C05453=1021.011,30.378,396.099,166.914,51.135,159.364
C05454=1021.017,30.627,396.085,166.917,51.129,159.363
C05455=1021.022,30.877,396.069,166.919,51.125,159.363
C05456=1021.028,31.126,396.055,166.923,51.119,159.362
C05457=1021.034,31.376,396.039,166.924,51.114,159.361
C05458=1021.040,31.626,396.024,166.928,51.109,159.361
C05459=1021.045,31.875,396.009,166.931,51.103,159.361
C05460=1021.051,32.124,395.993,166.933,51.098,159.360
C05461=1021.057,32.373,395.978,166.936,51.093,159.359
C05462=1021.062,32.623,395.962,166.938,51.088,159.359
C05463=1021.069,32.873,395.948,166.941,51.082,159.358
C05464=1021.074,33.122,395.932,166.944,51.077,159.358
C05465=1021.080,33.372,395.917,166.946,51.072,159.357
C05466=1021.086,33.621,395.901,166.949,51.066,159.357
C05467=1021.092,33.870,395.887,166.951,51.061,159.356
C05468=1021.098,34.120,395.871,166.954,51.056,159.356
C05469=1021.103,34.370,395.855,166.957,51.050,159.355
C05470=1021.109,34.619,395.841,166.959,51.045,159.355
C05471=1021.115,34.868,395.825,166.962,51.040,159.354
C05472=1021.121,35.117,395.810,166.964,51.035,159.353
C05473=1021.126,35.367,395.795,166.967,51.030,159.353
C05474=1021.133,35.617,395.780,166.970,51.024,159.352
C05475=1021.138,35.866,395.764,166.972,51.019,159.352
C05476=1021.144,36.116,395.748,166.975,51.013,159.351
C05477=1021.150,36.365,395.733,166.977,51.008,159.351
C05478=1021.156,36.615,395.718,166.980,51.002,159.350
C05479=1021.162,36.864,395.703,166.983,50.997,159.350
C05480=1021.168,37.113,395.687,166.985,50.992,159.349
C05481=1021.173,37.363,395.671,166.988,50.986,159.348
C05482=1021.178,37.613,395.656,166.990,50.982,159.348
C05483=1021.184,37.862,395.640,166.994,50.976,159.347
C05484=1021.191,38.112,395.625,166.996,50.972,159.347
C05485=1021.196,38.360,395.609,166.999,50.966,159.346
C05486=1021.202,38.610,395.593,167.001,50.961,159.346
C05487=1021.207,38.860,395.578,167.004,50.956,159.345
C05488=1021.213,39.110,395.562,167.007,50.950,159.345
C05489=1021.218,39.359,395.547,167.009,50.945,159.344
C05490=1021.225,39.608,395.531,167.012,50.940,159.344
C05491=1021.231,39.858,395.515,167.014,50.934,159.343
C05492=1021.236,40.107,395.499,167.017,50.929,159.343
C05493=1021.242,40.357,395.484,167.019,50.924,159.342
C05494=1021.247,40.606,395.468,167.022,50.918,159.341
C05495=1021.254,40.856,395.453,167.024,50.914,159.341
C05496=1021.259,41.105,395.438,167.027,50.908,159.340
C05497=1021.265,41.354,395.421,167.030,50.903,159.340
C05498=1021.271,41.604,395.406,167.033,50.898,159.339
C05499=1021.276,41.853,395.389,167.035,50.892,159.339
C05500=1021.282,42.102,395.375,167.038,50.887,159.338
C05501=1021.288,42.352,395.359,167.040,50.881,159.338
C05502=1021.294,42.602,395.343,167.043,50.876,159.337
C05503=1021.300,42.885,395.325,167.047,50.870,159.337
C05504=1021.306,43.169,395.306,167.049,50.864,159.336
C05505=1021.313,43.453,395.289,167.052,50.859,159.335
C05506=1021.319,43.737,395.270,167.055,50.853,159.335
C05507=1021.325,43.987,395.254,167.057,50.848,159.334
C05508=1021.330,44.235,395.238,167.060,50.843,159.334
C05509=1021.336,44.485,395.222,167.062,50.837,159.333
C05510=1021.342,44.735,395.207,167.065,50.832,159.333
C05511=1021.347,44.984,395.190,167.068,50.827,159.332
C05512=1021.353,45.234,395.174,167.071,50.822,159.332
C05513=1021.358,45.483,395.158,167.073,50.817,159.331
C05514=1021.364,45.732,395.142,167.076,50.812,159.330
C05515=1021.370,45.982,395.126,167.078,50.807,159.330
C05516=1021.376,46.232,395.110,167.081,50.801,159.329
C05517=1021.382,46.481,395.094,167.083,50.796,159.329
C05518=1021.387,46.730,395.078,167.086,50.791,159.328
C05519=1021.393,46.979,395.062,167.088,50.785,159.328
C05520=1021.399,47.229,395.046,167.091,50.780,159.327
C05521=1021.404,47.479,395.030,167.094,50.775,159.327
C05522=1021.410,47.728,395.013,167.096,50.770,159.326
C05523=1021.415,47.977,394.997,167.099,50.765,159.325
C05524=1021.421,48.227,394.982,167.102,50.760,159.325
C05525=1021.427,48.476,394.966,167.104,50.754,159.324
C05526=1021.433,48.725,394.949,167.107,50.749,159.324
C05527=1021.439,48.975,394.933,167.110,50.744,159.323
C05528=1021.444,49.225,394.918,167.112,50.738,159.323
C05529=1021.450,49.473,394.902,167.115,50.733,159.322
C05530=1021.455,49.723,394.885,167.117,50.728,159.322
C05531=1021.461,49.972,394.869,167.120,50.723,159.321
C05532=1021.467,50.222,394.852,167.122,50.718,159.321
C05533=1021.472,50.472,394.837,167.125,50.712,159.320
C05534=1021.478,50.721,394.821,167.127,50.707,159.319
C05535=1021.484,50.970,394.804,167.131,50.702,159.319
C05536=1021.490,51.220,394.788,167.132,50.697,159.318
C05537=1021.496,51.468,394.772,167.136,50.691,159.318
C05538=1021.502,51.718,394.756,167.139,50.686,159.317
C05539=1021.506,51.968,394.740,167.141,50.681,159.317
C05540=1021.512,52.217,394.723,167.144,50.675,159.316
C05541=1021.518,52.467,394.707,167.146,50.670,159.315
C05542=1021.524,52.716,394.691,167.149,50.665,159.315
C05543=1021.530,52.965,394.675,167.151,50.660,159.314
C05544=1021.536,53.215,394.658,167.154,50.654,159.314
C05545=1021.542,53.464,394.642,167.156,50.649,159.313
C05546=1021.548,53.714,394.627,167.159,50.644,159.313
C05547=1021.553,53.964,394.610,167.162,50.638,159.312
C05548=1021.559,54.213,394.594,167.164,50.633,159.312
C05549=1021.564,54.462,394.578,167.167,50.627,159.311
C05550=1021.570,54.711,394.561,167.169,50.623,159.310
C05551=1021.576,54.960,394.545,167.172,50.617,159.310
C05552=1021.582,55.210,394.529,167.174,50.612,159.309
C05553=1021.588,55.459,394.513,167.177,50.606,159.309
C05554=1021.593,55.709,394.496,167.180,50.601,159.308
C05555=1021.599,55.958,394.479,167.182,50.596,159.307
C05556=1021.605,56.207,394.463,167.185,50.590,159.307
C05557=1021.611,56.457,394.447,167.187,50.585,159.306
C05558=1021.617,56.706,394.431,167.191,50.580,159.306
C05559=1021.623,56.955,394.414,167.193,50.574,159.305
C05560=1021.629,57.205,394.398,167.196,50.569,159.305
C05561=1021.635,57.454,394.382,167.198,50.563,159.304
C05562=1021.640,57.704,394.365,167.200,50.558,159.303
C05563=1021.646,57.953,394.349,167.204,50.553,159.303
C05564=1021.652,58.202,394.333,167.206,50.547,159.302
C05565=1021.658,58.452,394.316,167.209,50.542,159.302
C05566=1021.664,58.701,394.300,167.212,50.536,159.301
C05567=1021.671,58.985,394.281,167.214,50.531,159.300
C05568=1021.677,59.270,394.263,167.217,50.525,159.300
C05569=1021.684,59.552,394.244,167.221,50.518,159.299
C05570=1021.691,59.836,394.226,167.224,50.512,159.299
C05571=1021.696,60.086,394.210,167.225,50.507,159.298
C05572=1021.702,60.335,394.193,167.229,50.502,159.297
C05573=1021.708,60.584,394.177,167.232,50.496,159.297
C05574=1021.714,60.834,394.160,167.233,50.490,159.296
C05575=1021.720,61.083,394.144,167.237,50.485,159.296
C05576=1021.725,61.333,394.128,167.240,50.479,159.295
C05577=1021.732,61.583,394.111,167.241,50.474,159.294
C05578=1021.738,61.831,394.094,167.245,50.469,159.294
C05579=1021.744,62.081,394.078,167.248,50.463,159.293
C05580=1021.749,62.330,394.061,167.250,50.458,159.293
C05581=1021.755,62.580,394.045,167.253,50.453,159.292
C05582=1021.761,62.829,394.028,167.254,50.447,159.291
C05583=1021.767,63.078,394.012,167.258,50.442,159.291
C05584=1021.773,63.328,393.995,167.261,50.436,159.290
C05585=1021.779,63.577,393.978,167.263,50.431,159.290
C05586=1021.785,63.826,393.962,167.266,50.426,159.289
C05587=1021.793,64.185,393.938,167.269,50.418,159.288
C05588=1021.801,64.542,393.913,167.273,50.410,159.287
C05589=1021.809,64.899,393.890,167.277,50.403,159.287
C05590=1021.817,65.257,393.866,167.281,50.396,159.286
C05591=1021.823,65.506,393.849,167.283,50.390,159.285
C05592=1021.829,65.755,393.832,167.286,50.385,159.285
C05593=1021.835,66.005,393.816,167.289,50.379,159.284
C05594=1021.841,66.254,393.798,167.291,50.375,159.283
C05595=1021.847,66.504,393.782,167.294,50.369,159.283
C05596=1021.852,66.753,393.765,167.296,50.364,159.282
C05597=1021.858,67.002,393.748,167.299,50.358,159.282
C05598=1021.863,67.252,393.731,167.301,50.353,159.281
C05599=1021.869,67.501,393.715,167.304,50.348,159.280
C05600=1021.875,67.750,393.697,167.307,50.343,159.280
C05601=1021.881,68.000,393.681,167.309,50.337,159.279
C05602=1021.886,68.249,393.663,167.312,50.331,159.279
C05603=1021.893,68.499,393.647,167.314,50.327,159.278
C05604=1021.898,68.748,393.630,167.318,50.322,159.278
C05605=1021.904,68.997,393.613,167.320,50.316,159.277
C05606=1021.909,69.247,393.596,167.323,50.311,159.276
C05607=1021.915,69.496,393.579,167.325,50.306,159.276
C05608=1021.921,69.745,393.562,167.328,50.300,159.275
C05609=1021.927,69.995,393.544,167.330,50.295,159.275
C05610=1021.932,70.244,393.527,167.333,50.290,159.274
C05611=1021.939,70.493,393.511,167.336,50.284,159.274
C05612=1021.944,70.743,393.494,167.338,50.279,159.273
C05613=1021.949,70.992,393.476,167.341,50.274,159.272
C05614=1021.955,71.241,393.460,167.343,50.269,159.272
C05615=1021.961,71.491,393.442,167.346,50.263,159.271
C05616=1021.967,71.741,393.425,167.349,50.258,159.271
C05617=1021.973,71.989,393.408,167.351,50.253,159.270
C05618=1021.978,72.238,393.391,167.354,50.248,159.269
C05619=1021.984,72.488,393.374,167.357,50.242,159.269
C05620=1021.989,72.737,393.356,167.359,50.237,159.268
C05621=1021.996,72.987,393.339,167.362,50.232,159.268
C05622=1022.001,73.236,393.322,167.365,50.227,159.267
C05623=1022.006,73.486,393.305,167.367,50.221,159.266
C05624=1022.013,73.735,393.288,167.370,50.216,159.266
C05625=1022.019,73.984,393.270,167.372,50.211,159.265
C05626=1022.024,74.234,393.253,167.375,50.205,159.265
C05627=1022.029,74.446,393.239,167.378,50.201,159.264
C05628=1022.034,74.658,393.224,167.380,50.196,159.264
C05629=1022.039,74.871,393.210,167.382,50.191,159.263
C05630=1022.044,75.083,393.195,167.384,50.188,159.263
C05631=1022.049,75.295,393.180,167.386,50.183,159.262
C05632=1022.054,75.508,393.165,167.388,50.178,159.262
C05633=1022.058,75.720,393.151,167.390,50.173,159.261
C05634=1022.063,75.933,393.136,167.393,50.169,159.261
C05635=1022.069,76.182,393.118,167.396,50.163,159.260
C05636=1022.075,76.431,393.102,167.398,50.159,159.260
C05637=1022.081,76.681,393.084,167.401,50.153,159.259
C05638=1022.087,76.930,393.067,167.403,50.148,159.258
C05639=1022.092,77.179,393.049,167.406,50.142,159.258
C05640=1022.097,77.429,393.032,167.409,50.138,159.257
C05641=1022.103,77.679,393.014,167.411,50.132,159.257
C05642=1022.109,77.928,392.997,167.414,50.127,159.256
C05643=1022.114,78.177,392.979,167.417,50.122,159.255
C05644=1022.120,78.426,392.962,167.420,50.116,159.255
C05645=1022.126,78.676,392.944,167.422,50.111,159.254
C05646=1022.131,78.925,392.927,167.425,50.106,159.254
C05647=1022.137,79.174,392.909,167.427,50.101,159.253
C05648=1022.143,79.424,392.891,167.430,50.096,159.253
C05649=1022.149,79.673,392.874,167.433,50.091,159.252
C05650=1022.155,79.922,392.857,167.435,50.085,159.252
C05651=1022.160,80.171,392.840,167.438,50.080,159.251
C05652=1022.166,80.421,392.822,167.441,50.075,159.250
C05653=1022.172,80.670,392.804,167.443,50.070,159.250
C05654=1022.177,80.919,392.787,167.446,50.064,159.249
C05655=1022.183,81.169,392.769,167.448,50.059,159.249
C05656=1022.189,81.418,392.751,167.451,50.054,159.248
C05657=1022.194,81.667,392.734,167.453,50.049,159.247
C05658=1022.200,81.916,392.716,167.456,50.043,159.247
C05659=1022.206,82.166,392.698,167.459,50.038,159.246
C05660=1022.211,82.415,392.681,167.461,50.033,159.246
C05661=1022.217,82.664,392.663,167.465,50.028,159.245
C05662=1022.223,82.914,392.646,167.467,50.022,159.244
C05663=1022.228,83.163,392.628,167.470,50.017,159.244
C05664=1022.234,83.412,392.611,167.472,50.012,159.243
C05665=1022.240,83.662,392.593,167.475,50.007,159.243
C05666=1022.245,83.911,392.575,167.478,50.001,159.242
C05667=1022.252,84.161,392.557,167.480,49.996,159.241
C05668=1022.257,84.410,392.540,167.483,49.991,159.241
C05669=1022.263,84.659,392.522,167.485,49.985,159.240
C05670=1022.269,84.909,392.504,167.488,49.980,159.240
C05671=1022.274,85.158,392.487,167.490,49.975,159.239
C05672=1022.280,85.407,392.469,167.494,49.970,159.239
C05673=1022.286,85.656,392.451,167.497,49.964,159.238
C05674=1022.291,85.906,392.434,167.499,49.959,159.237
C05675=1022.297,86.155,392.416,167.502,49.953,159.237
C05676=1022.303,86.404,392.398,167.504,49.948,159.236
C05677=1022.309,86.653,392.381,167.507,49.943,159.236
C05678=1022.315,86.903,392.363,167.510,49.937,159.235
C05679=1022.320,87.152,392.345,167.512,49.933,159.234
C05680=1022.326,87.402,392.327,167.515,49.927,159.234
C05681=1022.332,87.651,392.310,167.517,49.921,159.233
C05682=1022.338,87.899,392.291,167.520,49.916,159.233
C05683=1022.344,88.149,392.273,167.523,49.911,159.232
C05684=1022.349,88.398,392.256,167.526,49.906,159.231
C05685=1022.355,88.648,392.238,167.529,49.900,159.231
C05686=1022.361,88.897,392.220,167.530,49.895,159.230
C05687=1022.367,89.147,392.202,167.534,49.890,159.230
C05688=1022.372,89.396,392.184,167.537,49.884,159.229
C05689=1022.378,89.646,392.166,167.539,49.879,159.228
C05690=1022.383,89.895,392.149,167.542,49.874,159.228
C05691=1022.389,90.143,392.130,167.544,49.869,159.227
C05692=1022.395,90.393,392.112,167.547,49.863,159.227
C05693=1022.400,90.642,392.094,167.549,49.859,159.226
C05694=1022.406,90.892,392.076,167.552,49.853,159.225
C05695=1022.413,91.175,392.056,167.555,49.847,159.225
C05696=1022.419,91.459,392.035,167.558,49.841,159.224
C05697=1022.425,91.742,392.014,167.561,49.836,159.224
C05698=1022.432,92.026,391.993,167.565,49.829,159.223
C05699=1022.437,92.275,391.975,167.567,49.824,159.222
C05700=1022.443,92.525,391.957,167.570,49.819,159.222
C05701=1022.448,92.774,391.939,167.572,49.814,159.221
C05702=1022.455,93.023,391.921,167.575,49.808,159.221
C05703=1022.460,93.272,391.903,167.578,49.804,159.220
C05704=1022.466,93.522,391.885,167.581,49.798,159.219
C05705=1022.471,93.771,391.866,167.584,49.793,159.219
C05706=1022.477,94.020,391.849,167.586,49.787,159.218
C05707=1022.483,94.270,391.831,167.589,49.782,159.218
C05708=1022.488,94.518,391.812,167.591,49.777,159.217
C05709=1022.494,94.768,391.794,167.594,49.772,159.217
C05710=1022.500,95.016,391.776,167.596,49.767,159.216
C05711=1022.505,95.267,391.757,167.600,49.762,159.215
C05712=1022.511,95.516,391.739,167.603,49.756,159.215
C05713=1022.517,95.765,391.721,167.605,49.751,159.214
C05714=1022.523,96.015,391.702,167.608,49.746,159.214
C05715=1022.528,96.264,391.685,167.610,49.740,159.213
C05716=1022.535,96.513,391.666,167.613,49.735,159.212
C05717=1022.539,96.762,391.648,167.616,49.729,159.212
C05718=1022.546,97.011,391.629,167.618,49.725,159.211
C05719=1022.551,97.260,391.612,167.621,49.719,159.211
C05720=1022.557,97.510,391.592,167.624,49.714,159.210
C05721=1022.563,97.759,391.575,167.627,49.709,159.209
C05722=1022.569,98.009,391.557,167.630,49.703,159.209
C05723=1022.574,98.258,391.538,167.632,49.698,159.208
C05724=1022.580,98.507,391.520,167.635,49.693,159.207
C05725=1022.586,98.756,391.502,167.638,49.688,159.207
C05726=1022.591,99.006,391.483,167.640,49.682,159.206
C05727=1022.597,99.255,391.465,167.643,49.677,159.206
C05728=1022.603,99.504,391.447,167.645,49.672,159.205
C05729=1022.609,99.753,391.428,167.648,49.666,159.204
C05730=1022.614,100.003,391.409,167.652,49.661,159.204
C05731=1022.620,100.252,391.391,167.654,49.657,159.203
C05732=1022.626,100.501,391.372,167.657,49.651,159.203
C05733=1022.631,100.750,391.354,167.659,49.646,159.202
C05734=1022.637,101.000,391.335,167.662,49.640,159.202
C05735=1022.642,101.249,391.317,167.665,49.636,159.201
C05736=1022.648,101.498,391.298,167.668,49.630,159.200
C05737=1022.654,101.747,391.279,167.670,49.625,159.200
C05738=1022.659,101.997,391.261,167.673,49.620,159.199
C05739=1022.665,102.246,391.242,167.676,49.615,159.199
C05740=1022.670,102.495,391.223,167.678,49.609,159.198
C05741=1022.676,102.744,391.205,167.681,49.604,159.198
C05742=1022.682,102.994,391.186,167.683,49.599,159.197
C05743=1022.687,103.243,391.167,167.687,49.594,159.196
C05744=1022.693,103.492,391.149,167.690,49.588,159.196
C05745=1022.699,103.742,391.130,167.692,49.584,159.195
C05746=1022.704,103.990,391.112,167.695,49.578,159.195
C05747=1022.710,104.240,391.093,167.697,49.573,159.194
C05748=1022.715,104.489,391.074,167.700,49.568,159.193
C05749=1022.721,104.738,391.056,167.703,49.563,159.193
C05750=1022.727,104.988,391.036,167.706,49.557,159.192
C05751=1022.732,105.237,391.018,167.709,49.552,159.192
C05752=1022.738,105.486,391.000,167.711,49.547,159.191
C05753=1022.744,105.735,390.980,167.714,49.542,159.191
C05754=1022.750,105.984,390.962,167.717,49.536,159.190
C05755=1022.755,106.233,390.943,167.720,49.532,159.189
C05756=1022.761,106.483,390.924,167.723,49.526,159.189
C05757=1022.767,106.732,390.906,167.725,49.521,159.188
C05758=1022.772,106.981,390.887,167.728,49.516,159.188
C05759=1022.779,107.265,390.866,167.731,49.510,159.187
C05760=1022.785,107.549,390.845,167.735,49.504,159.186
C05761=1022.792,107.832,390.823,167.737,49.498,159.186
C05762=1022.799,108.116,390.801,167.740,49.492,159.185
C05763=1022.804,108.365,390.783,167.743,49.486,159.184
C05764=1022.810,108.614,390.764,167.746,49.482,159.184
C05765=1022.815,108.864,390.745,167.749,49.476,159.183
C05766=1022.821,109.113,390.727,167.752,49.471,159.183
C05767=1022.827,109.362,390.708,167.754,49.466,159.182
C05768=1022.833,109.612,390.688,167.757,49.460,159.181
C05769=1022.839,109.861,390.670,167.760,49.455,159.181
C05770=1022.844,110.109,390.651,167.762,49.450,159.180
C05771=1022.850,110.359,390.632,167.766,49.445,159.180
C05772=1022.856,110.608,390.612,167.769,49.439,159.179
C05773=1022.861,110.858,390.593,167.771,49.434,159.178
C05774=1022.867,111.106,390.575,167.774,49.429,159.178
C05775=1022.873,111.356,390.556,167.776,49.424,159.177
C05776=1022.878,111.605,390.536,167.779,49.419,159.177
C05777=1022.884,111.854,390.517,167.783,49.414,159.176
C05778=1022.889,112.103,390.498,167.785,49.408,159.175
C05779=1022.895,112.353,390.479,167.788,49.403,159.175
C05780=1022.901,112.602,390.460,167.791,49.398,159.174
C05781=1022.906,112.851,390.441,167.793,49.393,159.174
C05782=1022.911,113.100,390.422,167.797,49.388,159.173
C05783=1022.917,113.350,390.402,167.799,49.383,159.173
C05784=1022.923,113.599,390.383,167.802,49.378,159.172
C05785=1022.928,113.848,390.364,167.804,49.373,159.172
C05786=1022.933,114.097,390.345,167.807,49.367,159.171
C05787=1022.939,114.346,390.325,167.810,49.363,159.170
C05788=1022.945,114.595,390.306,167.813,49.358,159.170
C05789=1022.951,114.845,390.287,167.816,49.352,159.169
C05790=1022.956,115.094,390.268,167.818,49.348,159.169
C05791=1022.961,115.343,390.248,167.822,49.342,159.168
C05792=1022.967,115.593,390.229,167.824,49.337,159.168
C05793=1022.973,115.842,390.209,167.827,49.332,159.167
C05794=1022.978,116.091,390.189,167.830,49.327,159.166
C05795=1022.983,116.340,390.171,167.833,49.322,159.166
C05796=1022.989,116.589,390.151,167.836,49.317,159.165
C05797=1022.995,116.838,390.131,167.838,49.312,159.165
C05798=1023.001,117.087,390.112,167.841,49.307,159.164
C05799=1023.006,117.337,390.093,167.844,49.301,159.164
C05800=1023.011,117.586,390.073,167.847,49.297,159.163
C05801=1023.017,117.835,390.053,167.850,49.292,159.163
C05802=1023.022,118.084,390.034,167.852,49.286,159.162
C05803=1023.028,118.334,390.015,167.855,49.281,159.161
C05804=1023.034,118.583,389.996,167.858,49.276,159.161
C05805=1023.039,118.831,389.976,167.861,49.271,159.160
C05806=1023.045,119.081,389.957,167.864,49.265,159.160
C05807=1023.051,119.330,389.938,167.867,49.260,159.159
C05808=1023.056,119.579,389.918,167.869,49.256,159.159
C05809=1023.062,119.829,389.898,167.872,49.250,159.158
C05810=1023.067,120.078,389.879,167.876,49.245,159.157
C05811=1023.073,120.327,389.859,167.878,49.240,159.157
C05812=1023.078,120.576,389.840,167.881,49.235,159.156
C05813=1023.084,120.825,389.821,167.883,49.230,159.156
C05814=1023.090,121.074,389.801,167.887,49.225,159.155
C05815=1023.096,121.323,389.781,167.890,49.219,159.154
C05816=1023.101,121.573,389.762,167.892,49.215,159.154
C05817=1023.107,121.822,389.742,167.895,49.210,159.153
C05818=1023.112,122.071,389.722,167.898,49.204,159.153
C05819=1023.118,122.321,389.703,167.901,49.199,159.152
C05820=1023.124,122.569,389.683,167.904,49.194,159.152
C05821=1023.130,122.819,389.664,167.907,49.189,159.151
C05822=1023.135,123.068,389.645,167.910,49.183,159.150
C05823=1023.141,123.351,389.623,167.913,49.178,159.150
C05824=1023.148,123.635,389.600,167.916,49.172,159.149
C05825=1023.154,123.919,389.578,167.920,49.165,159.148
C05826=1023.161,124.202,389.556,167.923,49.160,159.148
C05827=1023.167,124.451,389.536,167.926,49.155,159.147
C05828=1023.172,124.701,389.516,167.928,49.150,159.147
C05829=1023.178,124.950,389.496,167.932,49.145,159.146
C05830=1023.184,125.199,389.477,167.935,49.139,159.146
C05831=1023.190,125.448,389.457,167.937,49.134,159.145
C05832=1023.195,125.697,389.437,167.940,49.129,159.144
C05833=1023.201,125.946,389.418,167.943,49.124,159.144
C05834=1023.207,126.196,389.398,167.947,49.118,159.143
C05835=1023.212,126.445,389.378,167.949,49.114,159.143
C05836=1023.218,126.694,389.358,167.952,49.108,159.142
C05837=1023.224,126.943,389.339,167.955,49.103,159.142
C05838=1023.230,127.192,389.319,167.957,49.098,159.141
C05839=1023.236,127.441,389.299,167.961,49.093,159.140
C05840=1023.241,127.691,389.280,167.964,49.087,159.140
C05841=1023.247,127.939,389.260,167.967,49.082,159.139
C05842=1023.252,128.189,389.240,167.969,49.077,159.139
C05843=1023.258,128.438,389.220,167.973,49.072,159.138
C05844=1023.264,128.687,389.201,167.976,49.067,159.137
C05845=1023.270,128.936,389.181,167.979,49.061,159.137
C05846=1023.276,129.186,389.162,167.981,49.056,159.136
C05847=1023.282,129.434,389.142,167.984,49.051,159.136
C05848=1023.288,129.683,389.122,167.987,49.046,159.135
C05849=1023.292,129.933,389.102,167.990,49.040,159.134
C05850=1023.298,130.182,389.082,167.993,49.036,159.134
C05851=1023.304,130.431,389.062,167.996,49.031,159.133
C05852=1023.309,130.680,389.042,167.999,49.025,159.133
C05853=1023.315,130.929,389.022,168.003,49.020,159.132
C05854=1023.321,131.178,389.002,168.005,49.015,159.132
C05855=1023.327,131.427,388.982,168.008,49.010,159.131
C05856=1023.332,131.677,388.962,168.011,49.005,159.131
C05857=1023.338,131.926,388.942,168.013,49.000,159.130
C05858=1023.343,132.175,388.922,168.017,48.995,159.129
C05859=1023.349,132.424,388.902,168.020,48.990,159.129
C05860=1023.354,132.673,388.881,168.022,48.985,159.128
C05861=1023.360,132.922,388.862,168.026,48.980,159.128
C05862=1023.365,133.171,388.841,168.029,48.974,159.127
C05863=1023.372,133.421,388.821,168.032,48.969,159.127
C05864=1023.377,133.670,388.800,168.034,48.965,159.126
C05865=1023.383,133.919,388.780,168.038,48.959,159.125
C05866=1023.388,134.168,388.760,168.041,48.954,159.125
C05867=1023.394,134.417,388.741,168.043,48.950,159.124
C05868=1023.399,134.666,388.720,168.046,48.944,159.124
C05869=1023.405,134.915,388.700,168.050,48.939,159.123
C05870=1023.410,135.164,388.680,168.053,48.934,159.123
C05871=1023.416,135.413,388.660,168.055,48.929,159.122
C05872=1023.422,135.662,388.639,168.059,48.924,159.122
C05873=1023.428,135.911,388.619,168.062,48.919,159.121
C05874=1023.433,136.161,388.598,168.065,48.914,159.121
C05875=1023.439,136.410,388.579,168.067,48.908,159.120
C05876=1023.444,136.659,388.558,168.071,48.903,159.119
C05877=1023.450,136.908,388.538,168.074,48.899,159.119
C05878=1023.456,137.157,388.518,168.077,48.893,159.118
C05879=1023.461,137.407,388.497,168.079,48.888,159.118
C05880=1023.467,137.655,388.477,168.083,48.884,159.117
C05881=1023.473,137.905,388.456,168.086,48.878,159.117
C05882=1023.479,138.154,388.436,168.089,48.873,159.116
C05883=1023.484,138.403,388.416,168.092,48.868,159.116
C05884=1023.489,138.652,388.395,168.095,48.863,159.115
C05885=1023.495,138.901,388.375,168.098,48.858,159.114
C05886=1023.500,139.150,388.355,168.101,48.853,159.114
C05887=1023.507,139.434,388.331,168.105,48.848,159.113
C05888=1023.513,139.718,388.307,168.108,48.842,159.113
C05889=1023.520,140.001,388.284,168.112,48.836,159.112
C05890=1023.526,140.284,388.261,168.115,48.831,159.111
C05891=1023.532,140.533,388.240,168.118,48.825,159.111
C05892=1023.537,140.782,388.219,168.121,48.820,159.110
C05893=1023.543,141.031,388.199,168.124,48.816,159.110
C05894=1023.549,141.281,388.179,168.127,48.810,159.109
C05895=1023.554,141.530,388.158,168.130,48.805,159.109
C05896=1023.559,141.779,388.137,168.134,48.800,159.108
C05897=1023.565,142.027,388.117,168.136,48.796,159.108
C05898=1023.571,142.276,388.096,168.139,48.790,159.107
C05899=1023.577,142.526,388.075,168.142,48.785,159.107
C05900=1023.582,142.775,388.055,168.146,48.780,159.106
C05901=1023.588,143.024,388.035,168.148,48.775,159.105
C05902=1023.593,143.273,388.013,168.151,48.770,159.105
C05903=1023.599,143.522,387.993,168.155,48.765,159.104
C05904=1023.605,143.772,387.972,168.158,48.760,159.104
C05905=1023.611,144.020,387.952,168.161,48.755,159.103
C05906=1023.616,144.269,387.931,168.164,48.750,159.103
C05907=1023.622,144.519,387.910,168.167,48.745,159.102
C05908=1023.627,144.768,387.889,168.170,48.740,159.102
C05909=1023.632,145.017,387.869,168.174,48.735,159.101
C05910=1023.639,145.265,387.848,168.177,48.730,159.100
C05911=1023.645,145.515,387.827,168.179,48.725,159.100
C05912=1023.650,145.764,387.807,168.182,48.720,159.099
C05913=1023.655,146.013,387.786,168.185,48.715,159.099
C05914=1023.661,146.262,387.764,168.189,48.710,159.098
C05915=1023.667,146.512,387.744,168.192,48.705,159.098
C05916=1023.672,146.760,387.723,168.195,48.700,159.097
C05917=1023.678,147.009,387.703,168.198,48.695,159.097
C05918=1023.684,147.259,387.682,168.201,48.690,159.096
C05919=1023.689,147.507,387.660,168.205,48.685,159.096
C05920=1023.695,147.756,387.640,168.208,48.680,159.095
C05921=1023.701,148.006,387.618,168.210,48.676,159.095
C05922=1023.706,148.255,387.598,168.214,48.670,159.094
C05923=1023.712,148.503,387.576,168.217,48.665,159.094
C05924=1023.717,148.752,387.556,168.220,48.660,159.093
C05925=1023.723,149.002,387.535,168.224,48.655,159.093
C05926=1023.728,149.251,387.514,168.226,48.650,159.092
C05927=1023.734,149.500,387.493,168.229,48.645,159.091
C05928=1023.740,149.749,387.472,168.233,48.641,159.091
C05929=1023.745,149.998,387.451,168.236,48.636,159.090
C05930=1023.751,150.247,387.430,168.240,48.631,159.090
C05931=1023.756,150.496,387.407,168.242,48.626,159.089
C05932=1023.761,150.745,387.387,168.245,48.621,159.089
C05933=1023.767,150.994,387.366,168.249,48.616,159.088
C05934=1023.773,151.244,387.345,168.252,48.611,159.088
C05935=1023.778,151.492,387.323,168.255,48.606,159.087
C05936=1023.784,151.742,387.303,168.258,48.601,159.087
C05937=1023.790,151.990,387.281,168.261,48.596,159.086
C05938=1023.795,152.240,387.261,168.264,48.591,159.086
C05939=1023.801,152.489,387.239,168.268,48.586,159.085
C05940=1023.807,152.737,387.218,168.271,48.581,159.085
C05941=1023.812,152.986,387.197,168.274,48.576,159.084
C05942=1023.818,153.236,387.176,168.278,48.571,159.084
C05943=1023.824,153.484,387.154,168.280,48.567,159.083
C05944=1023.830,153.734,387.133,168.284,48.562,159.083
C05945=1023.834,153.983,387.112,168.287,48.557,159.082
C05946=1023.841,154.232,387.090,168.290,48.551,159.081
C05947=1023.846,154.481,387.069,168.294,48.547,159.081
C05948=1023.851,154.730,387.048,168.297,48.542,159.080
C05949=1023.858,154.979,387.026,168.299,48.537,159.080
C05950=1023.862,155.228,387.005,168.303,48.532,159.079
C05951=1023.869,155.512,386.981,168.307,48.527,159.079
C05952=1023.875,155.794,386.956,168.310,48.521,159.078
C05953=1023.882,156.078,386.933,168.314,48.515,159.078
C05954=1023.888,156.360,386.908,168.317,48.510,159.077
C05955=1023.894,156.610,386.887,168.321,48.505,159.077
C05956=1023.899,156.858,386.865,168.324,48.500,159.076
C05957=1023.905,157.108,386.844,168.328,48.495,159.076
C05958=1023.910,157.357,386.823,168.331,48.490,159.075
C05959=1023.917,157.606,386.801,168.334,48.486,159.075
C05960=1023.921,157.855,386.779,168.338,48.480,159.074
C05961=1023.928,158.104,386.757,168.341,48.475,159.074
C05962=1023.933,158.352,386.736,168.343,48.471,159.073
C05963=1023.939,158.602,386.715,168.347,48.466,159.072
C05964=1023.945,158.851,386.694,168.350,48.461,159.072
C05965=1023.950,159.100,386.672,168.354,48.456,159.072
C05966=1023.956,159.349,386.650,168.357,48.451,159.071
C05967=1023.961,159.598,386.628,168.361,48.447,159.071
C05968=1023.967,159.847,386.607,168.364,48.442,159.070
C05969=1023.972,160.096,386.585,168.367,48.437,159.070
C05970=1023.977,160.345,386.563,168.370,48.432,159.069
C05971=1023.983,160.594,386.541,168.373,48.428,159.069
C05972=1023.988,160.843,386.519,168.377,48.423,159.068
C05973=1023.993,161.091,386.497,168.380,48.418,159.068
C05974=1023.999,161.341,386.475,168.383,48.413,159.067
C05975=1024.004,161.589,386.453,168.386,48.409,159.067
C05976=1024.009,161.839,386.431,168.390,48.404,159.066
C05977=1024.015,162.087,386.410,168.393,48.400,159.066
C05978=1024.020,162.337,386.388,168.397,48.395,159.065
C05979=1024.025,162.585,386.365,168.400,48.390,159.065
C05980=1024.032,162.834,386.343,168.403,48.385,159.064
C05981=1024.037,163.084,386.321,168.406,48.381,159.064
C05982=1024.042,163.333,386.299,168.410,48.376,159.063
C05983=1024.048,163.582,386.278,168.413,48.371,159.063
C05984=1024.053,163.831,386.256,168.417,48.366,159.062
C05985=1024.059,164.080,386.233,168.420,48.361,159.062
C05986=1024.064,164.328,386.212,168.423,48.357,159.061
C05987=1024.070,164.578,386.189,168.426,48.352,159.061
C05988=1024.074,164.826,386.167,168.429,48.347,159.060
C05989=1024.081,165.075,386.145,168.433,48.342,159.060
C05990=1024.086,165.325,386.123,168.436,48.338,159.059
C05991=1024.091,165.573,386.101,168.440,48.333,159.059
C05992=1024.097,165.823,386.079,168.443,48.329,159.059
C05993=1024.102,166.071,386.057,168.447,48.324,159.058
C05994=1024.108,166.320,386.035,168.450,48.319,159.058
C05995=1024.113,166.569,386.013,168.454,48.314,159.057
C05996=1024.119,166.818,385.990,168.457,48.309,159.057
C05997=1024.125,167.067,385.968,168.460,48.305,159.056
C05998=1024.130,167.316,385.947,168.463,48.300,159.056
C05999=1024.135,167.565,385.925,168.467,48.295,159.055
C06000=1024.141,167.814,385.902,168.470,48.290,159.055
C06001=1024.146,168.063,385.880,168.474,48.286,159.054
C06002=1024.153,168.311,385.857,168.477,48.281,159.054
C06003=1024.158,168.561,385.835,168.480,48.276,159.053
C06004=1024.163,168.810,385.813,168.484,48.271,159.053
C06005=1024.169,169.058,385.791,168.488,48.267,159.052
C06006=1024.175,169.308,385.769,168.491,48.262,159.052
C06007=1024.179,169.557,385.747,168.495,48.258,159.052
C06008=1024.186,169.805,385.725,168.498,48.253,159.051
C06009=1024.191,170.055,385.702,168.502,48.248,159.051
C06010=1024.197,170.303,385.680,168.505,48.243,159.050
C06011=1024.203,170.552,385.658,168.509,48.238,159.050
C06012=1024.208,170.802,385.636,168.512,48.234,159.049
C06013=1024.213,171.050,385.613,168.515,48.229,159.049
C06014=1024.219,171.299,385.591,168.519,48.224,159.048
C06015=1024.226,171.582,385.566,168.522,48.219,159.048
C06016=1024.232,171.865,385.540,168.527,48.213,159.047
C06017=1024.238,172.147,385.516,168.531,48.208,159.047
C06018=1024.245,172.431,385.490,168.534,48.203,159.046
C06019=1024.250,172.680,385.467,168.538,48.198,159.046
C06020=1024.256,172.928,385.445,168.541,48.193,159.045
C06021=1024.262,173.177,385.423,168.545,48.189,159.045
C06022=1024.267,173.426,385.400,168.548,48.184,159.044
C06023=1024.273,173.676,385.378,168.551,48.179,159.044
C06024=1024.279,173.924,385.356,168.555,48.174,159.043
C06025=1024.284,174.173,385.333,168.558,48.169,159.043
C06026=1024.290,174.422,385.311,168.563,48.164,159.042
C06027=1024.296,174.671,385.288,168.566,48.160,159.042
C06028=1024.302,174.920,385.266,168.570,48.155,159.041
C06029=1024.308,175.169,385.243,168.574,48.151,159.041
C06030=1024.312,175.418,385.221,168.577,48.146,159.040
C06031=1024.319,175.667,385.199,168.581,48.141,159.040
C06032=1024.325,175.915,385.176,168.584,48.136,159.040
C06033=1024.330,176.165,385.154,168.588,48.132,159.039
C06034=1024.336,176.414,385.132,168.591,48.127,159.039
C06035=1024.342,176.662,385.109,168.594,48.122,159.038
C06036=1024.347,176.911,385.087,168.598,48.117,159.038
C06037=1024.353,177.160,385.064,168.601,48.112,159.037
C06038=1024.359,177.409,385.041,168.605,48.108,159.037
C06039=1024.365,177.658,385.019,168.608,48.103,159.036
C06040=1024.370,177.907,384.996,168.613,48.098,159.036
C06041=1024.377,178.156,384.974,168.617,48.094,159.035
C06042=1024.382,178.405,384.952,168.620,48.089,159.035
C06043=1024.388,178.654,384.929,168.624,48.084,159.034
C06044=1024.393,178.902,384.906,168.627,48.079,159.034
C06045=1024.400,179.151,384.884,168.631,48.075,159.033
C06046=1024.405,179.400,384.862,168.634,48.070,159.033
C06047=1024.411,179.649,384.839,168.638,48.065,159.032
C06048=1024.416,179.898,384.816,168.641,48.060,159.032
C06049=1024.423,180.147,384.793,168.645,48.055,159.032
C06050=1024.428,180.396,384.771,168.649,48.051,159.031
C06051=1024.434,180.645,384.748,168.653,48.046,159.031
C06052=1024.440,180.894,384.725,168.656,48.042,159.030
C06053=1024.446,181.143,384.703,168.660,48.037,159.030
C06054=1024.452,181.392,384.680,168.663,48.032,159.029
C06055=1024.458,181.641,384.657,168.667,48.027,159.029
C06056=1024.464,181.890,384.635,168.671,48.022,159.028
C06057=1024.470,182.139,384.612,168.675,48.018,159.028
C06058=1024.475,182.388,384.589,168.678,48.013,159.027
C06059=1024.481,182.636,384.566,168.682,48.009,159.027
C06060=1024.486,182.886,384.543,168.685,48.004,159.027
C06061=1024.492,183.135,384.520,168.689,47.999,159.026
C06062=1024.498,183.383,384.497,168.693,47.995,159.026
C06063=1024.503,183.633,384.474,168.696,47.990,159.025
C06064=1024.509,183.881,384.450,168.700,47.986,159.025
C06065=1024.514,184.130,384.427,168.703,47.982,159.025
C06066=1024.519,184.379,384.403,168.707,47.977,159.024
C06067=1024.524,184.627,384.381,168.711,47.973,159.024
C06068=1024.530,184.876,384.358,168.716,47.968,159.024
C06069=1024.535,185.125,384.334,168.719,47.964,159.023
C06070=1024.541,185.374,384.311,168.723,47.959,159.023
C06071=1024.547,185.622,384.288,168.726,47.955,159.022
C06072=1024.552,185.872,384.264,168.730,47.950,159.022
C06073=1024.558,186.121,384.241,168.734,47.946,159.021
C06074=1024.563,186.369,384.217,168.737,47.941,159.021
C06075=1024.569,186.618,384.194,168.741,47.937,159.021
C06076=1024.574,186.867,384.171,168.744,47.932,159.020
C06077=1024.580,187.116,384.147,168.748,47.928,159.020
C06078=1024.585,187.364,384.124,168.752,47.923,159.019
C06079=1024.592,187.647,384.097,168.756,47.918,159.019
C06080=1024.598,187.930,384.071,168.761,47.913,159.019
C06081=1024.604,188.212,384.044,168.765,47.908,159.018
C06082=1024.611,188.494,384.018,168.769,47.903,159.018
C06083=1024.617,188.743,383.995,168.773,47.899,159.017
C06084=1024.622,188.992,383.970,168.777,47.894,159.017
C06085=1024.628,189.241,383.947,168.781,47.890,159.016
C06086=1024.633,189.490,383.924,168.784,47.885,159.016
C06087=1024.639,189.738,383.900,168.788,47.881,159.016
C06088=1024.645,189.987,383.877,168.792,47.876,159.015
C06089=1024.650,190.237,383.854,168.796,47.872,159.015
C06090=1024.656,190.485,383.830,168.800,47.867,159.014
C06091=1024.662,190.734,383.807,168.804,47.863,159.014
C06092=1024.667,190.982,383.783,168.807,47.858,159.014
C06093=1024.673,191.231,383.760,168.811,47.854,159.013
C06094=1024.679,191.481,383.735,168.815,47.849,159.013
C06095=1024.684,191.729,383.712,168.819,47.845,159.013
C06096=1024.690,191.978,383.689,168.823,47.841,159.012
C06097=1024.695,192.227,383.665,168.826,47.836,159.012
C06098=1024.701,192.475,383.641,168.830,47.832,159.011
C06099=1024.706,192.724,383.618,168.835,47.827,159.011
C06100=1024.713,192.973,383.594,168.838,47.823,159.010
C06101=1024.719,193.222,383.571,168.842,47.818,159.010
C06102=1024.724,193.471,383.547,168.846,47.814,159.010
C06103=1024.730,193.720,383.524,168.849,47.809,159.009
C06104=1024.735,193.968,383.499,168.854,47.805,159.009
C06105=1024.741,194.217,383.476,168.857,47.800,159.008
C06106=1024.747,194.466,383.452,168.861,47.796,159.008
C06107=1024.753,194.715,383.428,168.865,47.792,159.008
C06108=1024.758,194.964,383.405,168.870,47.787,159.007
C06109=1024.765,195.212,383.381,168.873,47.783,159.007
C06110=1024.770,195.462,383.358,168.877,47.778,159.007
C06111=1024.776,195.710,383.334,168.881,47.774,159.006
C06112=1024.781,195.959,383.310,168.885,47.769,159.006
C06113=1024.787,196.208,383.287,168.889,47.765,159.006
C06114=1024.793,196.457,383.262,168.893,47.760,159.005
C06115=1024.799,196.705,383.238,168.897,47.756,159.005
C06116=1024.805,196.954,383.215,168.901,47.751,159.004
C06117=1024.810,197.203,383.191,168.905,47.747,159.004
C06118=1024.817,197.452,383.167,168.908,47.743,159.003
C06119=1024.822,197.701,383.144,168.913,47.738,159.003
C06120=1024.828,197.949,383.120,168.917,47.733,159.003
C06121=1024.834,198.198,383.096,168.920,47.729,159.002
C06122=1024.840,198.447,383.072,168.925,47.725,159.002
C06123=1024.845,198.696,383.049,168.929,47.720,159.002
C06124=1024.851,198.945,383.024,168.933,47.716,159.001
C06125=1024.857,199.193,383.000,168.937,47.711,159.001
C06126=1024.863,199.441,382.977,168.941,47.707,159.001
C06127=1024.869,199.691,382.952,168.944,47.703,159.000
C06128=1024.875,199.940,382.929,168.949,47.698,159.000
C06129=1024.881,200.189,382.905,168.953,47.694,159.000
C06130=1024.886,200.438,382.880,168.957,47.690,158.999
C06131=1024.892,200.686,382.856,168.961,47.685,158.999
C06132=1024.898,200.935,382.832,168.965,47.681,158.998
C06133=1024.904,201.184,382.808,168.969,47.677,158.998
C06134=1024.909,201.432,382.784,168.973,47.672,158.998
C06135=1024.915,201.682,382.759,168.977,47.668,158.997
C06136=1024.920,201.930,382.735,168.981,47.664,158.997
C06137=1024.926,202.178,382.711,168.985,47.660,158.997
C06138=1024.932,202.428,382.686,168.990,47.656,158.996
C06139=1024.937,202.676,382.662,168.993,47.651,158.996
C06140=1024.943,202.925,382.637,168.997,47.647,158.996
C06141=1024.949,203.173,382.613,169.002,47.643,158.995
C06142=1024.955,203.422,382.589,169.006,47.639,158.995
C06143=1024.978,204.455,382.488,169.408,47.739,159.070
C06144=1024.990,204.861,382.446,169.413,47.733,159.069
C06145=1025.000,205.266,382.404,169.418,47.728,159.069
C06146=1025.011,205.671,382.362,169.422,47.723,159.068
C06147=1025.021,206.078,382.319,169.428,47.717,159.068
C06148=1025.028,206.326,382.293,169.431,47.714,159.068
C06149=1025.034,206.575,382.267,169.434,47.710,159.067
C06150=1025.041,206.823,382.241,169.438,47.706,159.067
C06151=1025.048,207.071,382.215,169.441,47.703,159.067
C06152=1025.054,207.321,382.189,169.444,47.700,159.067
C06153=1025.061,207.569,382.163,169.447,47.697,159.066
C06154=1025.067,207.817,382.138,169.450,47.693,159.066
C06155=1025.074,208.066,382.112,169.453,47.690,159.066
C06156=1025.080,208.314,382.085,169.456,47.687,159.065
C06157=1025.086,208.563,382.060,169.459,47.683,159.065
C06158=1025.093,208.812,382.033,169.463,47.680,159.065
C06159=1025.100,209.060,382.007,169.466,47.676,159.064
C06160=1025.106,209.308,381.981,169.469,47.673,159.064
C06161=1025.112,209.558,381.955,169.472,47.670,159.064
C06162=1025.119,209.806,381.929,169.475,47.666,159.064
C06163=1025.126,210.054,381.902,169.478,47.663,159.063
C06164=1025.132,210.303,381.877,169.481,47.660,159.063
C06165=1025.139,210.551,381.851,169.485,47.657,159.063
C06166=1025.145,210.800,381.824,169.488,47.653,159.062
C06167=1025.152,211.048,381.798,169.491,47.650,159.062
C06168=1025.158,211.297,381.771,169.494,47.647,159.062
C06169=1025.164,211.545,381.745,169.497,47.644,159.062
C06170=1025.171,211.794,381.720,169.500,47.641,159.061
C06171=1025.177,212.043,381.693,169.503,47.637,159.061
C06172=1025.184,212.291,381.666,169.506,47.634,159.061
C06173=1025.190,212.540,381.639,169.509,47.631,159.061
C06174=1025.196,212.788,381.613,169.513,47.628,159.060
C06175=1025.203,213.036,381.587,169.516,47.624,159.060
C06176=1025.209,213.285,381.560,169.520,47.621,159.060
C06177=1025.216,213.533,381.534,169.523,47.618,159.060
C06178=1025.223,213.782,381.508,169.526,47.615,159.059
C06179=1025.229,214.030,381.481,169.529,47.611,159.059
C06180=1025.236,214.279,381.455,169.532,47.608,159.059
C06181=1025.242,214.528,381.428,169.535,47.605,159.058
C06182=1025.248,214.777,381.402,169.538,47.602,159.058
C06183=1025.255,215.025,381.376,169.542,47.599,159.058
C06184=1025.261,215.274,381.349,169.545,47.596,159.058
C06185=1025.268,215.522,381.323,169.548,47.593,159.058
C06186=1025.274,215.771,381.296,169.551,47.590,159.057
C06187=1025.281,216.019,381.270,169.554,47.587,159.057
C06188=1025.288,216.268,381.244,169.558,47.583,159.057
C06189=1025.294,216.516,381.217,169.560,47.580,159.056
C06190=1025.301,216.765,381.191,169.564,47.576,159.056
C06191=1025.307,217.013,381.163,169.568,47.573,159.056
C06192=1025.314,217.262,381.137,169.571,47.570,159.056
C06193=1025.320,217.510,381.111,169.574,47.567,159.056
C06194=1025.327,217.759,381.084,169.577,47.564,159.055
C06195=1025.333,218.007,381.058,169.580,47.561,159.055
C06196=1025.340,218.256,381.031,169.583,47.558,159.055
C06197=1025.346,218.504,381.005,169.587,47.555,159.055
C06198=1025.353,218.753,380.978,169.590,47.551,159.054
C06199=1025.359,219.001,380.952,169.593,47.548,159.054
C06200=1025.371,219.409,380.907,169.599,47.543,159.054
C06201=1025.381,219.818,380.862,169.604,47.539,159.053
C06202=1025.391,220.226,380.819,169.609,47.534,159.053
C06203=1025.402,220.634,380.775,169.615,47.528,159.053
C06204=1025.408,220.882,380.748,169.618,47.525,159.052
C06205=1025.414,221.131,380.721,169.621,47.523,159.052
C06206=1025.421,221.379,380.694,169.624,47.520,159.052
C06207=1025.427,221.628,380.667,169.628,47.517,159.052
C06208=1025.434,221.877,380.640,169.631,47.514,159.052
C06209=1025.441,222.124,380.614,169.634,47.511,159.051
C06210=1025.447,222.373,380.587,169.638,47.507,159.051
C06211=1025.453,222.622,380.560,169.641,47.505,159.051
C06212=1025.460,222.870,380.533,169.644,47.502,159.051
C06213=1025.467,223.119,380.506,169.648,47.499,159.051
C06214=1025.473,223.367,380.478,169.651,47.496,159.050
C06215=1025.479,223.616,380.451,169.654,47.493,159.050
C06216=1025.486,223.864,380.425,169.657,47.490,159.050
C06217=1025.492,224.112,380.398,169.660,47.487,159.050
C06218=1025.499,224.361,380.371,169.664,47.484,159.050
C06219=1025.505,224.609,380.344,169.668,47.481,159.049
C06220=1025.512,224.858,380.317,169.671,47.478,159.049
C06221=1025.518,225.107,380.290,169.674,47.475,159.049
C06222=1025.525,225.354,380.263,169.677,47.472,159.049
C06223=1025.531,225.603,380.236,169.680,47.469,159.049
C06224=1025.538,225.852,380.208,169.684,47.467,159.048
C06225=1025.544,226.101,380.181,169.688,47.463,159.048
C06226=1025.551,226.348,380.155,169.691,47.460,159.048
C06227=1025.558,226.597,380.128,169.694,47.457,159.048
C06228=1025.564,226.846,380.100,169.698,47.455,159.048
C06229=1025.571,227.094,380.074,169.701,47.452,159.047
C06230=1025.578,227.342,380.046,169.704,47.449,159.047
C06231=1025.584,227.591,380.018,169.707,47.446,159.047
C06232=1025.590,227.839,379.992,169.710,47.443,159.047
C06233=1025.597,228.088,379.964,169.714,47.440,159.047
C06234=1025.603,228.337,379.937,169.718,47.438,159.047
C06235=1025.610,228.585,379.909,169.721,47.434,159.046
C06236=1025.616,228.833,379.882,169.724,47.432,159.046
C06237=1025.622,229.082,379.855,169.728,47.429,159.046
C06238=1025.629,229.330,379.827,169.731,47.427,159.046
C06239=1025.635,229.578,379.800,169.734,47.424,159.046
C06240=1025.642,229.827,379.772,169.737,47.420,159.046
C06241=1025.649,230.075,379.746,169.741,47.418,159.045
C06242=1025.655,230.324,379.718,169.745,47.415,159.045
C06243=1025.661,230.571,379.690,169.748,47.412,159.045
C06244=1025.668,230.820,379.663,169.751,47.409,159.045
C06245=1025.675,231.069,379.636,169.755,47.407,159.045
C06246=1025.680,231.318,379.607,169.758,47.404,159.045
C06247=1025.687,231.565,379.580,169.761,47.401,159.045
C06248=1025.693,231.814,379.552,169.765,47.399,159.044
C06249=1025.700,232.062,379.525,169.768,47.396,159.044
C06250=1025.706,232.311,379.498,169.771,47.394,159.044
C06251=1025.713,232.560,379.470,169.775,47.390,159.044
C06252=1025.719,232.808,379.442,169.779,47.388,159.044
C06253=1025.726,233.056,379.415,169.782,47.385,159.044
C06254=1025.732,233.304,379.387,169.785,47.382,159.044
C06255=1025.739,233.553,379.359,169.789,47.380,159.043
C06256=1025.749,233.953,379.314,169.795,47.375,159.043
C06257=1025.760,234.354,379.270,169.799,47.371,159.043
C06258=1025.770,234.754,379.225,169.805,47.367,159.043
C06259=1025.780,235.155,379.181,169.811,47.362,159.043
C06260=1025.786,235.403,379.153,169.815,47.360,159.042
C06261=1025.793,235.652,379.125,169.818,47.357,159.042
C06262=1025.800,235.900,379.098,169.821,47.354,159.042
C06263=1025.806,236.149,379.070,169.825,47.352,159.042
C06264=1025.813,236.397,379.042,169.828,47.349,159.042
C06265=1025.820,236.645,379.014,169.832,47.346,159.042
C06266=1025.826,236.893,378.986,169.835,47.344,159.042
C06267=1025.833,237.141,378.959,169.839,47.341,159.042
C06268=1025.839,237.390,378.930,169.842,47.338,159.041
C06269=1025.846,237.638,378.903,169.845,47.336,159.041
C06270=1025.852,237.887,378.875,169.849,47.334,159.041
C06271=1025.859,238.135,378.847,169.852,47.330,159.041
C06272=1025.866,238.384,378.819,169.856,47.328,159.041
C06273=1025.871,238.632,378.791,169.860,47.325,159.041
C06274=1025.878,238.881,378.763,169.863,47.323,159.041
C06275=1025.885,239.129,378.735,169.866,47.320,159.041
C06276=1025.892,239.377,378.707,169.870,47.318,159.041
C06277=1025.899,239.625,378.679,169.873,47.315,159.040
C06278=1025.904,239.874,378.651,169.877,47.313,159.040
C06279=1025.911,240.122,378.624,169.881,47.310,159.040
C06280=1025.918,240.370,378.595,169.885,47.308,159.040
C06281=1025.923,240.619,378.567,169.888,47.305,159.040
C06282=1025.930,240.867,378.539,169.891,47.302,159.040
C06283=1025.936,241.115,378.510,169.895,47.300,159.040
C06284=1025.943,241.364,378.482,169.898,47.297,159.040
C06285=1025.949,241.612,378.454,169.901,47.295,159.040
C06286=1025.956,241.860,378.426,169.905,47.293,159.040
C06287=1025.963,242.109,378.398,169.909,47.290,159.040
C06288=1025.969,242.357,378.369,169.913,47.288,159.040
C06289=1025.976,242.605,378.341,169.916,47.285,159.039
C06290=1025.982,242.854,378.313,169.920,47.283,159.039
C06291=1025.989,243.102,378.284,169.923,47.280,159.039
C06292=1025.995,243.350,378.256,169.926,47.278,159.039
C06293=1026.001,243.598,378.228,169.930,47.276,159.039
C06294=1026.007,243.847,378.199,169.933,47.273,159.039
C06295=1026.014,244.095,378.171,169.938,47.271,159.039
C06296=1026.020,244.344,378.142,169.941,47.268,159.039
C06297=1026.027,244.592,378.113,169.945,47.266,159.039
C06298=1026.033,244.840,378.086,169.948,47.263,159.039
C06299=1026.040,245.088,378.057,169.951,47.261,159.039
C06300=1026.046,245.336,378.028,169.955,47.259,159.039
C06301=1026.052,245.585,378.000,169.958,47.256,159.039
C06302=1026.059,245.833,377.971,169.962,47.255,159.039
C06303=1026.065,246.082,377.943,169.966,47.252,159.039
C06304=1026.071,246.330,377.913,169.970,47.249,159.039
C06305=1026.078,246.578,377.885,169.973,47.247,159.039
C06306=1026.084,246.826,377.857,169.977,47.245,159.038
C06307=1026.090,247.075,377.828,169.980,47.242,159.038
C06308=1026.097,247.322,377.799,169.984,47.241,159.038
C06309=1026.103,247.571,377.771,169.987,47.238,159.038
C06310=1026.109,247.819,377.742,169.991,47.236,159.038
C06311=1026.116,248.067,377.713,169.994,47.233,159.038
C06312=1026.126,248.462,377.667,170.000,47.230,159.038
C06313=1026.136,248.856,377.621,170.007,47.226,159.038
C06314=1026.147,249.251,377.576,170.012,47.223,159.038
C06315=1026.157,249.644,377.530,170.018,47.219,159.038
C06316=1026.163,249.893,377.502,170.022,47.217,159.038
C06317=1026.170,250.141,377.473,170.025,47.214,159.038
C06318=1026.177,250.390,377.444,170.028,47.212,159.038
C06319=1026.183,250.638,377.415,170.032,47.210,159.038
C06320=1026.189,250.886,377.386,170.036,47.208,159.038
C06321=1026.196,251.134,377.357,170.040,47.205,159.038
C06322=1026.202,251.382,377.329,170.044,47.203,159.038
C06323=1026.209,251.631,377.300,170.047,47.201,159.038
C06324=1026.215,251.879,377.271,170.051,47.199,159.038
C06325=1026.222,252.127,377.242,170.054,47.196,159.038
C06326=1026.228,252.375,377.213,170.058,47.194,159.038
C06327=1026.235,252.624,377.184,170.062,47.192,159.038
C06328=1026.241,252.872,377.155,170.066,47.189,159.038
C06329=1026.248,253.120,377.126,170.069,47.188,159.038
C06330=1026.255,253.368,377.097,170.073,47.185,159.038
C06331=1026.261,253.616,377.068,170.076,47.183,159.038
C06332=1026.267,253.865,377.039,170.081,47.181,159.038
C06333=1026.275,254.113,377.010,170.085,47.178,159.038
C06334=1026.281,254.361,376.981,170.088,47.176,159.038
C06335=1026.287,254.609,376.952,170.092,47.174,159.038
C06336=1026.294,254.858,376.923,170.095,47.172,159.038
C06337=1026.301,255.106,376.894,170.100,47.169,159.038
C06338=1026.307,255.354,376.865,170.103,47.168,159.038
C06339=1026.314,255.602,376.836,170.107,47.165,159.038
C06340=1026.320,255.851,376.807,170.110,47.163,159.038
C06341=1026.327,256.099,376.778,170.114,47.161,159.038
C06342=1026.334,256.347,376.749,170.118,47.158,159.038
C06343=1026.341,256.596,376.720,170.122,47.157,159.038
C06344=1026.347,256.844,376.691,170.126,47.154,159.038
C06345=1026.354,257.092,376.663,170.129,47.153,159.038
C06346=1026.361,257.341,376.633,170.133,47.150,159.038
C06347=1026.367,257.588,376.603,170.137,47.148,159.038
C06348=1026.373,257.836,376.574,170.141,47.146,159.038
C06349=1026.380,258.085,376.545,170.145,47.144,159.038
C06350=1026.387,258.333,376.516,170.148,47.142,159.038
C06351=1026.394,258.581,376.487,170.152,47.139,159.038
C06352=1026.400,258.830,376.458,170.156,47.137,159.038
C06353=1026.407,259.077,376.428,170.160,47.135,159.038
C06354=1026.415,259.326,376.399,170.163,47.133,159.038
C06355=1026.421,259.574,376.370,170.168,47.131,159.038
C06356=1026.427,259.822,376.341,170.172,47.129,159.038
C06357=1026.434,260.070,376.311,170.175,47.127,159.038
C06358=1026.441,260.318,376.283,170.179,47.125,159.038
C06359=1026.448,260.567,376.253,170.183,47.122,159.038
C06360=1026.454,260.815,376.224,170.187,47.120,159.038
C06361=1026.461,261.063,376.195,170.191,47.119,159.038
C06362=1026.468,261.312,376.165,170.194,47.116,159.038
C06363=1026.474,261.559,376.135,170.198,47.115,159.038
C06364=1026.480,261.808,376.105,170.203,47.113,159.038
C06365=1026.487,262.056,376.076,170.206,47.111,159.038
C06366=1026.493,262.304,376.047,170.210,47.108,159.038
C06367=1026.500,262.552,376.017,170.213,47.107,159.038
C06368=1026.510,262.945,375.969,170.220,47.104,159.038
C06369=1026.521,263.338,375.922,170.226,47.100,159.039
C06370=1026.531,263.730,375.876,170.232,47.097,159.039
C06371=1026.542,264.123,375.829,170.238,47.094,159.039
C06372=1026.548,264.371,375.799,170.242,47.093,159.039
C06373=1026.555,264.619,375.769,170.246,47.091,159.039
C06374=1026.561,264.868,375.739,170.251,47.089,159.039
C06375=1026.568,265.116,375.709,170.254,47.086,159.039
C06376=1026.575,265.363,375.680,170.258,47.085,159.039
C06377=1026.581,265.612,375.650,170.261,47.083,159.039
C06378=1026.587,265.860,375.620,170.265,47.081,159.039
C06379=1026.595,266.108,375.590,170.270,47.079,159.039
C06380=1026.601,266.356,375.561,170.274,47.078,159.040
C06381=1026.607,266.605,375.530,170.277,47.076,159.040
C06382=1026.614,266.852,375.500,170.281,47.074,159.040
C06383=1026.621,267.100,375.470,170.286,47.072,159.040
C06384=1026.627,267.348,375.440,170.289,47.070,159.040
C06385=1026.634,267.597,375.410,170.293,47.068,159.040
C06386=1026.640,267.845,375.381,170.297,47.066,159.040
C06387=1026.647,268.093,375.350,170.302,47.064,159.040
C06388=1026.653,268.341,375.320,170.305,47.063,159.040
C06389=1026.660,268.589,375.290,170.309,47.061,159.040
C06390=1026.666,268.837,375.260,170.313,47.059,159.040
C06391=1026.673,269.085,375.230,170.318,47.057,159.041
C06392=1026.680,269.334,375.200,170.321,47.055,159.041
C06393=1026.686,269.582,375.170,170.325,47.054,159.041
C06394=1026.693,269.830,375.140,170.329,47.052,159.041
C06395=1026.700,270.077,375.110,170.333,47.050,159.041
C06396=1026.706,270.326,375.079,170.337,47.048,159.041
C06397=1026.713,270.574,375.049,170.341,47.046,159.041
C06398=1026.719,270.822,375.019,170.345,47.045,159.041
C06399=1026.726,271.070,374.989,170.350,47.043,159.042
C06400=1026.732,271.318,374.958,170.353,47.042,159.042
C06401=1026.739,271.566,374.928,170.357,47.040,159.042
C06402=1026.746,271.814,374.897,170.361,47.038,159.042
C06403=1026.752,272.062,374.867,170.366,47.036,159.042
C06404=1026.759,272.310,374.836,170.369,47.035,159.042
C06405=1026.766,272.558,374.806,170.373,47.033,159.042
C06406=1026.772,272.806,374.776,170.377,47.032,159.042
C06407=1026.779,273.054,374.746,170.382,47.030,159.043
C06408=1026.785,273.303,374.715,170.386,47.028,159.043
C06409=1026.792,273.550,374.684,170.389,47.026,159.043
C06410=1026.799,273.798,374.654,170.393,47.025,159.043
C06411=1026.805,274.047,374.623,170.398,47.023,159.043
C06412=1026.812,274.294,374.593,170.402,47.021,159.043
C06413=1026.818,274.543,374.562,170.406,47.020,159.043
C06414=1026.825,274.791,374.531,170.410,47.019,159.044
C06415=1026.831,275.038,374.501,170.414,47.017,159.044
C06416=1026.838,275.287,374.471,170.418,47.015,159.044
C06417=1026.845,275.534,374.440,170.422,47.013,159.044
C06418=1026.852,275.783,374.409,170.427,47.012,159.044
C06419=1026.858,276.031,374.379,170.431,47.010,159.044
C06420=1026.865,276.278,374.348,170.434,47.008,159.044
C06421=1026.871,276.527,374.317,170.439,47.007,159.045
C06422=1026.879,276.775,374.287,170.443,47.005,159.045
C06423=1026.885,277.022,374.256,170.447,47.004,159.045
C06424=1026.896,277.420,374.206,170.454,47.001,159.045
C06425=1026.906,277.818,374.157,170.461,46.999,159.046
C06426=1026.916,278.215,374.108,170.467,46.996,159.046
C06427=1026.928,278.612,374.058,170.474,46.994,159.046
C06428=1026.933,278.860,374.028,170.478,46.992,159.046
C06429=1026.940,279.108,373.996,170.482,46.991,159.047
C06430=1026.947,279.356,373.965,170.486,46.990,159.047
C06431=1026.953,279.604,373.934,170.491,46.988,159.047
C06432=1026.960,279.852,373.903,170.495,46.987,159.047
C06433=1026.967,280.100,373.873,170.499,46.986,159.047
C06434=1026.973,280.348,373.842,170.503,46.984,159.048
C06435=1026.980,280.596,373.810,170.507,46.982,159.048
C06436=1026.986,280.844,373.779,170.511,46.981,159.048
C06437=1026.993,281.092,373.748,170.516,46.979,159.048
C06438=1027.000,281.340,373.717,170.520,46.978,159.048
C06439=1027.006,281.588,373.686,170.524,46.977,159.049
C06440=1027.012,281.836,373.655,170.528,46.976,159.049
C06441=1027.020,282.083,373.624,170.533,46.974,159.049
C06442=1027.027,282.331,373.592,170.537,46.972,159.049
C06443=1027.033,282.580,373.562,170.541,46.971,159.049
C06444=1027.040,282.828,373.530,170.546,46.969,159.050
C06445=1027.047,283.075,373.499,170.550,46.968,159.050
C06446=1027.053,283.323,373.467,170.553,46.967,159.050
C06447=1027.060,283.571,373.436,170.558,46.965,159.050
C06448=1027.067,283.820,373.406,170.563,46.964,159.051
C06449=1027.074,284.067,373.374,170.567,46.962,159.051
C06450=1027.081,284.315,373.343,170.571,46.961,159.051
C06451=1027.087,284.563,373.312,170.575,46.960,159.051
C06452=1027.094,284.811,373.280,170.580,46.958,159.051
C06453=1027.101,285.059,373.249,170.584,46.957,159.052
C06454=1027.107,285.307,373.217,170.588,46.956,159.052
C06455=1027.114,285.555,373.186,170.593,46.954,159.052
C06456=1027.121,285.803,373.154,170.597,46.953,159.052
C06457=1027.128,286.051,373.123,170.601,46.952,159.053
C06458=1027.134,286.299,373.092,170.606,46.950,159.053
C06459=1027.141,286.546,373.060,170.610,46.949,159.053
C06460=1027.148,286.794,373.029,170.615,46.947,159.053
C06461=1027.155,287.042,372.997,170.619,46.946,159.054
C06462=1027.161,287.290,372.966,170.623,46.945,159.054
C06463=1027.168,287.538,372.934,170.628,46.944,159.054
C06464=1027.175,287.786,372.903,170.632,46.943,159.054
C06465=1027.181,288.034,372.872,170.636,46.942,159.055
C06466=1027.188,288.282,372.840,170.641,46.940,159.055
C06467=1027.194,288.529,372.807,170.645,46.939,159.055
C06468=1027.201,288.777,372.776,170.649,46.938,159.056
C06469=1027.208,289.025,372.745,170.654,46.936,159.056
C06470=1027.215,289.273,372.713,170.658,46.935,159.056
C06471=1027.222,289.520,372.681,170.663,46.934,159.056
C06472=1027.228,289.769,372.649,170.667,46.933,159.057
C06473=1027.234,290.016,372.617,170.671,46.932,159.057
C06474=1027.241,290.264,372.586,170.676,46.930,159.057
C06475=1027.249,290.512,372.554,170.680,46.929,159.057
C06476=1027.255,290.760,372.522,170.685,46.928,159.058
C06477=1027.262,291.008,372.491,170.689,46.927,159.058
C06478=1027.268,291.256,372.458,170.693,46.926,159.058
C06479=1027.275,291.504,372.426,170.698,46.924,159.059
C06480=1027.287,291.914,372.374,170.706,46.923,159.059
C06481=1027.297,292.323,372.321,170.713,46.921,159.060
C06482=1027.309,292.732,372.268,170.721,46.919,159.060
C06483=1027.320,293.142,372.215,170.728,46.917,159.061
C06484=1027.327,293.390,372.183,170.732,46.916,159.061
C06485=1027.334,293.638,372.151,170.737,46.915,159.061
C06486=1027.340,293.885,372.119,170.741,46.914,159.062
C06487=1027.347,294.133,372.087,170.746,46.913,159.062
C06488=1027.353,294.381,372.054,170.750,46.912,159.062
C06489=1027.361,294.629,372.022,170.754,46.911,159.062
C06490=1027.367,294.877,371.990,170.760,46.910,159.063
C06491=1027.373,295.124,371.957,170.764,46.909,159.063
C06492=1027.380,295.372,371.925,170.769,46.908,159.064
C06493=1027.387,295.619,371.892,170.773,46.907,159.064
C06494=1027.393,295.868,371.860,170.777,46.906,159.064
C06495=1027.400,296.116,371.828,170.783,46.905,159.065
C06496=1027.406,296.363,371.795,170.787,46.904,159.065
C06497=1027.414,296.610,371.763,170.792,46.903,159.065
C06498=1027.420,296.858,371.730,170.796,46.902,159.066
C06499=1027.426,297.107,371.698,170.800,46.901,159.066
C06500=1027.433,297.354,371.665,170.805,46.901,159.066
C06501=1027.440,297.602,371.633,170.809,46.900,159.067
C06502=1027.447,297.850,371.600,170.814,46.898,159.067
C06503=1027.454,298.097,371.567,170.819,46.898,159.068
C06504=1027.460,298.345,371.535,170.824,46.896,159.068
C06505=1027.466,298.593,371.502,170.828,46.896,159.068
C06506=1027.474,298.841,371.469,170.832,46.895,159.069
C06507=1027.480,299.088,371.437,170.838,46.894,159.069
C06508=1027.486,299.336,371.404,170.842,46.893,159.069
C06509=1027.494,299.584,371.371,170.847,46.892,159.070
C06510=1027.500,299.831,371.339,170.851,46.891,159.070
C06511=1027.507,300.080,371.306,170.856,46.891,159.071
C06512=1027.514,300.327,371.273,170.860,46.890,159.071
C06513=1027.521,300.574,371.241,170.866,46.889,159.071
C06514=1027.527,300.823,371.208,170.870,46.888,159.072
C06515=1027.535,301.070,371.175,170.875,46.887,159.072
C06516=1027.541,301.318,371.143,170.879,46.887,159.072
C06517=1027.548,301.566,371.110,170.884,46.885,159.073
C06518=1027.555,301.813,371.077,170.889,46.885,159.073
C06519=1027.562,302.061,371.044,170.894,46.884,159.074
C06520=1027.568,302.308,371.011,170.898,46.883,159.074
C06521=1027.576,302.556,370.978,170.904,46.882,159.074
C06522=1027.582,302.804,370.946,170.908,46.881,159.075
C06523=1027.589,303.052,370.913,170.913,46.880,159.075
C06524=1027.596,303.299,370.879,170.917,46.880,159.076
C06525=1027.603,303.547,370.847,170.922,46.879,159.076
C06526=1027.610,303.795,370.814,170.927,46.878,159.076
C06527=1027.616,304.043,370.781,170.932,46.878,159.077
C06528=1027.624,304.290,370.748,170.936,46.877,159.077
C06529=1027.631,304.538,370.715,170.941,46.876,159.078
C06530=1027.637,304.786,370.682,170.946,46.875,159.078
C06531=1027.645,305.033,370.649,170.951,46.875,159.079
C06532=1027.651,305.281,370.616,170.955,46.873,159.079
C06533=1027.658,305.529,370.583,170.960,46.873,159.079
C06534=1027.665,305.776,370.550,170.966,46.872,159.080
C06535=1027.672,306.024,370.517,170.970,46.872,159.080
C06536=1027.679,306.237,370.488,170.974,46.871,159.081
C06537=1027.684,306.451,370.459,170.978,46.870,159.081
C06538=1027.690,306.664,370.431,170.983,46.870,159.081
C06539=1027.696,306.877,370.402,170.987,46.869,159.082
C06540=1027.703,307.091,370.374,170.991,46.868,159.082
C06541=1027.709,307.304,370.346,170.995,46.868,159.083
C06542=1027.715,307.518,370.317,171.000,46.867,159.083
C06543=1027.721,307.731,370.289,171.004,46.866,159.083
C06544=1027.728,307.978,370.255,171.008,46.866,159.084
C06545=1027.734,308.226,370.222,171.014,46.865,159.084
C06546=1027.742,308.474,370.189,171.019,46.864,159.085
C06547=1027.749,308.721,370.156,171.023,46.864,159.085
C06548=1027.756,308.969,370.122,171.029,46.863,159.086
C06549=1027.764,309.216,370.089,171.033,46.863,159.086
C06550=1027.771,309.465,370.056,171.038,46.862,159.087
C06551=1027.777,309.712,370.022,171.044,46.861,159.087
C06552=1027.784,309.959,369.989,171.048,46.861,159.087
C06553=1027.792,310.207,369.956,171.053,46.860,159.088
C06554=1027.799,310.455,369.922,171.059,46.859,159.088
C06555=1027.806,310.702,369.889,171.063,46.859,159.089
C06556=1027.813,310.950,369.856,171.068,46.858,159.089
C06557=1027.820,311.198,369.822,171.073,46.858,159.090
C06558=1027.827,311.445,369.788,171.078,46.857,159.090
C06559=1027.833,311.693,369.754,171.083,46.856,159.091
C06560=1027.840,311.941,369.720,171.088,46.856,159.091
C06561=1027.847,312.188,369.687,171.093,46.856,159.092
C06562=1027.854,312.435,369.653,171.098,46.855,159.092
C06563=1027.861,312.683,369.618,171.103,46.854,159.093
C06564=1027.868,312.931,369.585,171.108,46.855,159.093
C06565=1027.875,313.177,369.550,171.113,46.854,159.094
C06566=1027.881,313.425,369.516,171.118,46.853,159.094
C06567=1027.888,313.673,369.482,171.123,46.853,159.095
C06568=1027.895,313.921,369.448,171.128,46.853,159.096
C06569=1027.902,314.169,369.414,171.134,46.852,159.096
C06570=1027.909,314.416,369.380,171.138,46.852,159.097
C06571=1027.916,314.663,369.347,171.144,46.851,159.097
C06572=1027.923,314.911,369.312,171.148,46.852,159.098
C06573=1027.930,315.158,369.278,171.154,46.851,159.098
C06574=1027.937,315.406,369.244,171.159,46.850,159.099
C06575=1027.943,315.654,369.209,171.164,46.850,159.099
C06576=1027.950,315.901,369.176,171.169,46.850,159.100
C06577=1027.957,316.148,369.141,171.174,46.849,159.101
C06578=1027.964,316.396,369.107,171.179,46.849,159.101
C06579=1027.971,316.644,369.073,171.184,46.849,159.102
C06580=1027.978,316.891,369.038,171.190,46.848,159.102
C06581=1027.985,317.139,369.004,171.194,46.848,159.103
C06582=1027.992,317.386,368.970,171.200,46.848,159.103
C06583=1027.999,317.634,368.935,171.205,46.848,159.104
C06584=1028.006,317.881,368.901,171.210,46.847,159.104
C06585=1028.014,318.128,368.867,171.215,46.847,159.105
C06586=1028.020,318.376,368.833,171.221,46.846,159.105
C06587=1028.027,318.624,368.799,171.225,46.846,159.106
C06588=1028.035,318.871,368.764,171.231,46.846,159.107
C06589=1028.041,319.119,368.730,171.236,46.846,159.107
C06590=1028.049,319.366,368.695,171.241,46.846,159.108
C06591=1028.055,319.614,368.661,171.246,46.845,159.108
C06592=1028.063,319.861,368.626,171.252,46.845,159.109
C06593=1028.070,320.109,368.592,171.258,46.845,159.110
C06594=1028.077,320.356,368.557,171.262,46.844,159.110
C06595=1028.084,320.604,368.523,171.268,46.844,159.111
C06596=1028.091,320.820,368.493,171.272,46.844,159.111
C06597=1028.097,321.036,368.463,171.277,46.844,159.112
C06598=1028.103,321.252,368.433,171.282,46.843,159.112
C06599=1028.109,321.468,368.403,171.287,46.843,159.113
C06600=1028.115,321.683,368.373,171.291,46.843,159.113
C06601=1028.122,321.900,368.342,171.296,46.843,159.114
C06602=1028.128,322.114,368.312,171.300,46.843,159.114
C06603=1028.134,322.331,368.281,171.304,46.843,159.115
C06604=1028.142,322.579,368.248,171.310,46.843,159.116
C06605=1028.149,322.826,368.213,171.315,46.842,159.116
C06606=1028.156,323.074,368.178,171.321,46.842,159.117
C06607=1028.164,323.321,368.144,171.326,46.842,159.117
C06608=1028.170,323.569,368.109,171.331,46.842,159.118
C06609=1028.178,323.816,368.074,171.337,46.842,159.119
C06610=1028.185,324.063,368.040,171.343,46.842,159.120
C06611=1028.193,324.311,368.004,171.348,46.841,159.120
C06612=1028.200,324.558,367.970,171.354,46.841,159.121
C06613=1028.207,324.806,367.935,171.358,46.841,159.121
C06614=1028.215,325.054,367.900,171.364,46.841,159.122
C06615=1028.222,325.301,367.866,171.370,46.841,159.123
C06616=1028.229,325.548,367.831,171.375,46.841,159.123
C06617=1028.237,325.795,367.796,171.381,46.841,159.124
C06618=1028.244,326.043,367.760,171.386,46.840,159.125
C06619=1028.252,326.290,367.726,171.391,46.841,159.125
C06620=1028.260,326.538,367.691,171.397,46.841,159.126
C06621=1028.266,326.785,367.656,171.402,46.840,159.127
C06622=1028.274,327.032,367.621,171.408,46.840,159.127
C06623=1028.281,327.280,367.586,171.414,46.840,159.128
C06624=1028.289,327.528,367.551,171.419,46.840,159.129
C06625=1028.296,327.775,367.516,171.425,46.840,159.129
C06626=1028.303,328.023,367.481,171.430,46.840,159.130
C06627=1028.311,328.269,367.445,171.435,46.840,159.131
C06628=1028.318,328.517,367.410,171.441,46.841,159.131
C06629=1028.325,328.765,367.375,171.447,46.840,159.132
C06630=1028.332,329.012,367.339,171.452,46.840,159.133
C06631=1028.339,329.260,367.303,171.458,46.840,159.133
C06632=1028.346,329.507,367.268,171.463,46.841,159.134
C06633=1028.353,329.754,367.232,171.469,46.841,159.135
C06634=1028.361,330.002,367.198,171.474,46.841,159.136
C06635=1028.368,330.249,367.162,171.480,46.841,159.136
C06636=1028.376,330.496,367.126,171.486,46.841,159.137
C06637=1028.383,330.744,367.091,171.492,46.841,159.138
C06638=1028.390,330.991,367.055,171.497,46.842,159.139
C06639=1028.397,331.238,367.020,171.503,46.841,159.139
C06640=1028.405,331.486,366.984,171.509,46.841,159.140
C06641=1028.412,331.733,366.949,171.514,46.842,159.141
C06642=1028.420,331.980,366.913,171.519,46.842,159.141
C06643=1028.427,332.228,366.878,171.525,46.842,159.142
C06644=1028.434,332.475,366.841,171.531,46.842,159.143
C06645=1028.441,332.723,366.806,171.537,46.843,159.144
C06646=1028.449,332.970,366.770,171.543,46.843,159.144
C06647=1028.457,333.217,366.734,171.548,46.843,159.145
C06648=1028.464,333.465,366.699,171.554,46.843,159.146
C06649=1028.472,333.712,366.663,171.560,46.844,159.147
C06650=1028.479,333.959,366.627,171.566,46.843,159.148
C06651=1028.486,334.206,366.591,171.572,46.844,159.148
C06652=1028.494,334.454,366.555,171.577,46.844,159.149
C06653=1028.501,334.701,366.520,171.583,46.844,159.150
C06654=1028.508,334.948,366.483,171.589,46.845,159.151
C06655=1028.515,335.195,366.447,171.595,46.845,159.151
C06656=1028.522,335.410,366.416,171.600,46.846,159.152
C06657=1028.528,335.623,366.385,171.604,46.846,159.153
C06658=1028.534,335.837,366.354,171.609,46.846,159.153
C06659=1028.541,336.050,366.322,171.615,46.846,159.154
C06660=1028.547,336.264,366.291,171.620,46.846,159.155
C06661=1028.554,336.477,366.260,171.624,46.847,159.156
C06662=1028.560,336.691,366.228,171.630,46.847,159.156
C06663=1028.566,336.905,366.197,171.635,46.847,159.157
C06664=1028.574,337.152,366.161,171.641,46.848,159.158
C06665=1028.581,337.399,366.125,171.647,46.848,159.159
C06666=1028.589,337.646,366.089,171.653,46.849,159.160
C06667=1028.597,337.894,366.053,171.659,46.849,159.160
C06668=1028.603,338.142,366.016,171.664,46.849,159.161
C06669=1028.611,338.388,365.980,171.670,46.850,159.162
C06670=1028.618,338.636,365.944,171.676,46.850,159.163
C06671=1028.626,338.883,365.907,171.682,46.851,159.164
C06672=1028.634,339.130,365.871,171.688,46.851,159.164
C06673=1028.642,339.377,365.835,171.694,46.852,159.165
C06674=1028.649,339.625,365.798,171.700,46.852,159.166
C06675=1028.656,339.872,365.762,171.706,46.853,159.167
C06676=1028.664,340.119,365.725,171.712,46.853,159.168
C06677=1028.671,340.366,365.689,171.718,46.853,159.169
C06678=1028.679,340.614,365.653,171.724,46.854,159.170
C06679=1028.687,340.860,365.616,171.731,46.854,159.171
C06680=1028.694,341.108,365.579,171.737,46.855,159.171
C06681=1028.702,341.355,365.542,171.742,46.855,159.172
C06682=1028.709,341.603,365.505,171.749,46.856,159.173
C06683=1028.716,341.849,365.468,171.755,46.857,159.174
C06684=1028.724,342.096,365.432,171.761,46.857,159.175
C06685=1028.731,342.343,365.395,171.767,46.858,159.176
C06686=1028.739,342.591,365.359,171.772,46.858,159.177
C06687=1028.747,342.838,365.322,171.779,46.859,159.178
C06688=1028.754,343.086,365.285,171.785,46.860,159.179
C06689=1028.762,343.332,365.248,171.791,46.860,159.179
C06690=1028.769,343.579,365.210,171.798,46.860,159.180
C06691=1028.777,343.827,365.174,171.804,46.862,159.181
C06692=1028.784,344.074,365.137,171.810,46.862,159.182
C06693=1028.792,344.321,365.100,171.816,46.863,159.183
C06694=1028.799,344.568,365.063,171.822,46.864,159.184
C06695=1028.807,344.815,365.026,171.828,46.864,159.185
C06696=1028.815,345.062,364.989,171.834,46.865,159.186
C06697=1028.822,345.309,364.951,171.841,46.865,159.187
C06698=1028.830,345.556,364.915,171.847,46.866,159.188
C06699=1028.837,345.805,364.877,171.853,46.867,159.189
C06700=1028.845,346.052,364.840,171.859,46.867,159.190
C06701=1028.853,346.299,364.803,171.865,46.869,159.191
C06702=1028.861,346.546,364.766,171.871,46.869,159.192
C06703=1028.868,346.793,364.728,171.879,46.870,159.193
C06704=1028.876,347.039,364.691,171.885,46.870,159.194
C06705=1028.883,347.287,364.654,171.891,46.871,159.195
C06706=1028.892,347.534,364.617,171.897,46.872,159.196
C06707=1028.899,347.781,364.579,171.903,46.873,159.196
C06708=1028.907,348.028,364.542,171.910,46.874,159.198
C06709=1028.915,348.275,364.505,171.916,46.874,159.198
C06710=1028.922,348.522,364.468,171.923,46.875,159.199
C06711=1028.930,348.770,364.430,171.929,46.876,159.200
C06712=1028.938,349.016,364.392,171.936,46.877,159.201
C06713=1028.945,349.263,364.355,171.942,46.878,159.202
C06714=1028.953,349.510,364.317,171.948,46.879,159.203
C06715=1028.961,349.758,364.279,171.954,46.880,159.205
C06716=1028.967,349.970,364.247,171.960,46.880,159.205
C06717=1028.974,350.181,364.215,171.965,46.881,159.206
C06718=1028.981,350.393,364.182,171.972,46.882,159.207
C06719=1028.987,350.606,364.150,171.977,46.883,159.208
C06720=1028.994,350.817,364.118,171.982,46.883,159.209
C06721=1029.001,351.030,364.086,171.989,46.884,159.210
C06722=1029.007,351.242,364.053,171.994,46.885,159.211
C06723=1029.014,351.454,364.020,172.000,46.886,159.212
C06724=1029.021,351.701,363.982,172.006,46.887,159.213
C06725=1029.029,351.947,363.944,172.012,46.888,159.214
C06726=1029.038,352.195,363.907,172.019,46.889,159.215
C06727=1029.045,352.441,363.869,172.026,46.890,159.216
C06728=1029.053,352.689,363.831,172.032,46.891,159.217
C06729=1029.060,352.936,363.793,172.039,46.891,159.218
C06730=1029.068,353.183,363.756,172.045,46.893,159.219
C06731=1029.077,353.430,363.717,172.052,46.894,159.220
C06732=1029.084,353.676,363.679,172.059,46.895,159.221
C06733=1029.092,353.924,363.641,172.065,46.896,159.222
C06734=1029.100,354.170,363.603,172.072,46.897,159.223
C06735=1029.108,354.418,363.565,172.079,46.898,159.224
C06736=1029.116,354.665,363.527,172.085,46.899,159.225
C06737=1029.124,354.912,363.488,172.091,46.900,159.227
C06738=1029.132,355.158,363.451,172.099,46.901,159.228
C06739=1029.140,355.405,363.412,172.105,46.903,159.229
C06740=1029.148,355.652,363.374,172.113,46.903,159.230
C06741=1029.156,355.900,363.336,172.119,46.904,159.231
C06742=1029.163,356.146,363.298,172.125,46.906,159.232
C06743=1029.171,356.393,363.259,172.133,46.907,159.233
C06744=1029.180,356.641,363.221,172.139,46.908,159.234
C06745=1029.187,356.887,363.182,172.146,46.909,159.236
C06746=1029.195,357.134,363.144,172.153,46.910,159.237
C06747=1029.203,357.381,363.106,172.160,46.912,159.238
C06748=1029.211,357.628,363.067,172.166,46.913,159.239
C06749=1029.219,357.875,363.028,172.174,46.914,159.240
C06750=1029.227,358.121,362.989,172.180,46.915,159.241
C06751=1029.235,358.368,362.951,172.188,46.917,159.243
C06752=1029.243,358.616,362.912,172.194,46.918,159.244
C06753=1029.251,358.862,362.874,172.201,46.919,159.245
C06754=1029.259,359.109,362.835,172.208,46.920,159.246
C06755=1029.267,359.356,362.796,172.214,46.922,159.247
C06756=1029.276,359.603,362.757,172.222,46.923,159.248
C06757=1029.283,359.850,362.719,172.229,46.924,159.250
C06758=1029.292,360.096,362.680,172.236,46.926,159.251
C06759=1029.300,360.344,362.641,172.243,46.926,159.252
C06760=1029.308,360.591,362.603,172.250,46.928,159.253
C06761=1029.316,360.837,362.564,172.257,46.929,159.254
C06762=1029.324,361.084,362.525,172.264,46.931,159.256
C06763=1029.332,361.331,362.485,172.271,46.932,159.257
C06764=1029.340,361.578,362.446,172.278,46.933,159.258
C06765=1029.348,361.825,362.407,172.285,46.935,159.259
C06766=1029.356,362.071,362.368,172.292,46.937,159.261
C06767=1029.363,362.318,362.329,172.299,46.938,159.262
C06768=1029.372,362.565,362.290,172.307,46.939,159.263
C06769=1029.380,362.811,362.250,172.313,46.941,159.264
C06770=1029.389,363.058,362.212,172.321,46.942,159.266
C06771=1029.396,363.305,362.172,172.328,46.944,159.267
C06772=1029.405,363.552,362.132,172.335,46.945,159.268
C06773=1029.413,363.798,362.094,172.343,46.947,159.269
C06774=1029.420,364.045,362.054,172.349,46.948,159.271
C06775=1029.428,364.292,362.015,172.357,46.950,159.272
C06776=1029.438,364.577,361.969,172.365,46.952,159.273
C06777=1029.447,364.861,361.924,172.374,46.953,159.275
C06778=1029.457,365.146,361.878,172.382,46.955,159.276
C06779=1029.466,365.430,361.832,172.390,46.957,159.278
C06780=1029.475,365.677,361.793,172.398,46.958,159.279
C06781=1029.483,365.924,361.754,172.405,46.960,159.280
C06782=1029.491,366.170,361.714,172.412,46.962,159.282
C06783=1029.500,366.417,361.674,172.420,46.963,159.283
C06784=1029.508,366.664,361.635,172.427,46.965,159.284
C06785=1029.516,366.910,361.596,172.434,46.966,159.286
C06786=1029.525,367.158,361.556,172.442,46.968,159.287
C06787=1029.533,367.404,361.516,172.450,46.970,159.289
C06788=1029.542,367.651,361.477,172.456,46.972,159.290
C06789=1029.550,367.897,361.436,172.464,46.973,159.291
C06790=1029.558,368.144,361.397,172.472,46.975,159.293
C06791=1029.567,368.391,361.358,172.479,46.976,159.294
C06792=1029.575,368.638,361.317,172.486,46.978,159.295
C06793=1029.584,368.884,361.277,172.494,46.980,159.297
C06794=1029.592,369.131,361.238,172.501,46.981,159.298
C06795=1029.600,369.378,361.198,172.509,46.983,159.299
C06796=1029.614,369.770,361.134,172.521,46.986,159.302
C06797=1029.627,370.162,361.069,172.533,46.989,159.304
C06798=1029.640,370.555,361.006,172.546,46.992,159.306
C06799=1029.653,370.947,360.941,172.558,46.995,159.308
C06800=1029.662,371.193,360.901,172.566,46.997,159.310
C06801=1029.670,371.441,360.861,172.572,46.999,159.311
C06802=1029.678,371.687,360.820,172.580,47.001,159.313
C06803=1029.687,371.933,360.780,172.588,47.003,159.314
C06804=1029.695,372.180,360.739,172.596,47.004,159.316
C06805=1029.704,372.427,360.700,172.604,47.006,159.317
C06806=1029.712,372.673,360.659,172.612,47.008,159.319
C06807=1029.721,372.920,360.618,172.619,47.010,159.320
C06808=1029.729,373.166,360.578,172.627,47.012,159.322
C06809=1029.738,373.413,360.537,172.635,47.014,159.323
C06810=1029.746,373.659,360.497,172.643,47.016,159.324
C06811=1029.755,373.906,360.456,172.651,47.018,159.326
C06812=1029.763,374.152,360.416,172.659,47.019,159.327
C06813=1029.771,374.398,360.375,172.666,47.022,159.329
C06814=1029.781,374.645,360.335,172.674,47.024,159.331
C06815=1029.789,374.892,360.294,172.682,47.026,159.332
C06816=1029.797,375.138,360.253,172.690,47.028,159.334
C06817=1029.807,375.385,360.213,172.698,47.030,159.335
C06818=1029.815,375.631,360.172,172.705,47.032,159.336
C06819=1029.823,375.878,360.131,172.715,47.034,159.338
C06820=1029.832,376.124,360.090,172.723,47.036,159.340
C06821=1029.841,376.371,360.049,172.730,47.038,159.341
C06822=1029.850,376.618,360.008,172.739,47.040,159.343
C06823=1029.859,376.863,359.968,172.747,47.042,159.344
C06824=1029.867,377.110,359.927,172.754,47.044,159.346
C06825=1029.876,377.357,359.886,172.763,47.047,159.347
C06826=1029.885,377.602,359.845,172.771,47.049,159.349
C06827=1029.894,377.849,359.804,172.779,47.051,159.351
C06828=1029.903,378.096,359.762,172.787,47.053,159.352
C06829=1029.911,378.342,359.721,172.795,47.056,159.354
C06830=1029.920,378.588,359.680,172.803,47.057,159.355
C06831=1029.929,378.835,359.638,172.811,47.060,159.357
C06832=1029.936,379.060,359.600,172.819,47.062,159.358
C06833=1029.944,379.287,359.563,172.827,47.064,159.360
C06834=1029.952,379.512,359.525,172.834,47.067,159.362
C06835=1029.960,379.738,359.487,172.842,47.068,159.363
C06836=1029.968,379.964,359.449,172.850,47.070,159.365
C06837=1029.976,380.189,359.411,172.857,47.072,159.366
C06838=1029.984,380.416,359.372,172.864,47.074,159.367
C06839=1029.992,380.641,359.335,172.873,47.077,159.369
C06840=1030.001,380.887,359.293,172.881,47.079,159.371
C06841=1030.010,381.134,359.251,172.889,47.081,159.372
C06842=1030.019,381.380,359.209,172.897,47.084,159.374
C06843=1030.028,381.627,359.168,172.905,47.086,159.376
C06844=1030.037,381.873,359.126,172.914,47.088,159.377
C06845=1030.046,382.119,359.084,172.923,47.091,159.379
C06846=1030.054,382.366,359.043,172.931,47.093,159.381
C06847=1030.063,382.612,359.001,172.939,47.096,159.382
C06848=1030.072,382.858,358.959,172.948,47.098,159.384
C06849=1030.081,383.104,358.916,172.956,47.100,159.386
C06850=1030.090,383.351,358.874,172.965,47.104,159.388
C06851=1030.099,383.597,358.833,172.974,47.106,159.389
C06852=1030.108,383.844,358.791,172.982,47.108,159.391
C06853=1030.117,384.089,358.749,172.991,47.111,159.393
C06854=1030.126,384.336,358.707,173.000,47.113,159.395
C06855=1030.135,384.582,358.665,173.008,47.116,159.396
C06856=1030.144,384.828,358.623,173.017,47.118,159.398
C06857=1030.153,385.074,358.581,173.026,47.120,159.400
C06858=1030.162,385.320,358.539,173.034,47.124,159.402
C06859=1030.172,385.567,358.496,173.044,47.126,159.403
C06860=1030.181,385.813,358.455,173.052,47.128,159.405
C06861=1030.190,386.059,358.412,173.061,47.131,159.407
C06862=1030.199,386.305,358.371,173.070,47.133,159.409
C06863=1030.208,386.551,358.328,173.078,47.136,159.411
C06864=1030.218,386.798,358.285,173.087,47.139,159.412
C06865=1030.227,387.044,358.244,173.096,47.142,159.414
C06866=1030.236,387.290,358.201,173.105,47.144,159.416
C06867=1030.245,387.536,358.158,173.114,47.147,159.418
C06868=1030.254,387.782,358.115,173.123,47.150,159.420
C06869=1030.264,388.028,358.073,173.132,47.153,159.422
C06870=1030.272,388.275,358.031,173.141,47.155,159.424
C06871=1030.282,388.521,357.988,173.149,47.158,159.425
C06872=1030.291,388.767,357.945,173.159,47.160,159.427
C06873=1030.300,389.013,357.903,173.167,47.164,159.429
C06874=1030.309,389.259,357.860,173.177,47.166,159.431
C06875=1030.319,389.505,357.817,173.187,47.169,159.433
C06876=1030.328,389.751,357.774,173.195,47.172,159.435
C06877=1030.337,389.997,357.731,173.205,47.175,159.437
C06878=1030.346,390.243,357.688,173.213,47.178,159.439
C06879=1030.356,390.489,357.645,173.223,47.180,159.441
C06880=1030.365,390.735,357.602,173.232,47.183,159.443
C06881=1030.375,390.981,357.559,173.241,47.186,159.444
C06882=1030.383,391.227,357.516,173.250,47.189,159.446
C06883=1030.393,391.473,357.473,173.260,47.192,159.448
C06884=1030.402,391.719,357.429,173.269,47.195,159.450
C06885=1030.412,391.965,357.386,173.278,47.198,159.452
C06886=1030.421,392.211,357.343,173.288,47.201,159.454
C06887=1030.431,392.457,357.300,173.297,47.204,159.456
C06888=1030.440,392.703,357.256,173.306,47.207,159.458
C06889=1030.449,392.949,357.213,173.316,47.210,159.460
C06890=1030.459,393.195,357.169,173.326,47.213,159.462
C06891=1030.468,393.442,357.126,173.334,47.216,159.464
C06892=1030.478,393.684,357.084,173.344,47.219,159.466
C06893=1030.487,393.928,357.040,173.354,47.222,159.468
C06894=1030.496,394.172,356.997,173.362,47.225,159.470
C06895=1030.506,394.415,356.954,173.372,47.228,159.472
C06896=1030.515,394.658,356.911,173.382,47.231,159.475
C06897=1030.524,394.902,356.867,173.391,47.234,159.476
C06898=1030.534,395.146,356.825,173.400,47.238,159.479
C06899=1030.544,395.389,356.781,173.410,47.241,159.481
C06900=1030.553,395.636,356.737,173.420,47.244,159.483
C06901=1030.563,395.881,356.693,173.430,47.247,159.485
C06902=1030.572,396.128,356.649,173.439,47.250,159.487
C06903=1030.581,396.373,356.606,173.449,47.253,159.489
C06904=1030.592,396.618,356.561,173.459,47.257,159.491
C06905=1030.601,396.864,356.517,173.469,47.260,159.493
C06906=1030.611,397.110,356.473,173.479,47.263,159.495
C06907=1030.621,397.356,356.430,173.489,47.266,159.498
C06908=1030.630,397.602,356.385,173.499,47.270,159.500
C06909=1030.640,397.848,356.341,173.509,47.273,159.502
C06910=1030.650,398.094,356.297,173.519,47.276,159.504
C06911=1030.659,398.340,356.253,173.528,47.279,159.506
C06912=1030.669,398.585,356.208,173.538,47.283,159.508
C06913=1030.679,398.831,356.165,173.548,47.287,159.511
C06914=1030.689,399.077,356.120,173.558,47.290,159.513
C06915=1030.698,399.323,356.076,173.568,47.293,159.515
C06916=1030.708,399.568,356.031,173.578,47.297,159.517
C06917=1030.718,399.814,355.987,173.588,47.300,159.519
C06918=1030.729,400.060,355.942,173.598,47.303,159.522
C06919=1030.738,400.306,355.897,173.608,47.307,159.524
C06920=1030.748,400.551,355.853,173.618,47.310,159.526
C06921=1030.757,400.798,355.808,173.629,47.314,159.528
C06922=1030.767,401.043,355.764,173.640,47.318,159.531
C06923=1030.777,401.289,355.719,173.650,47.321,159.533
C06924=1030.788,401.535,355.674,173.660,47.325,159.535
C06925=1030.798,401.780,355.629,173.670,47.328,159.538
C06926=1030.807,402.026,355.585,173.680,47.332,159.540
C06927=1030.818,402.272,355.539,173.691,47.335,159.542
C06928=1030.827,402.517,355.495,173.701,47.339,159.545
C06929=1030.837,402.763,355.450,173.712,47.343,159.547
C06930=1030.847,403.009,355.405,173.722,47.347,159.549
C06931=1030.856,403.255,355.359,173.733,47.350,159.552
C06932=1030.866,403.500,355.314,173.743,47.354,159.554
C06933=1030.877,403.746,355.268,173.753,47.358,159.556
C06934=1030.886,403.991,355.224,173.764,47.361,159.559
C06935=1030.897,404.237,355.178,173.775,47.365,159.561
C06936=1030.907,404.483,355.133,173.785,47.369,159.564
C06937=1030.917,404.729,355.088,173.796,47.372,159.566
C06938=1030.927,404.974,355.042,173.807,47.376,159.568
C06939=1030.937,405.220,354.997,173.817,47.380,159.571
C06940=1030.947,405.465,354.951,173.828,47.384,159.573
C06941=1030.958,405.711,354.906,173.839,47.387,159.576
C06942=1030.968,405.956,354.861,173.850,47.391,159.578
C06943=1030.978,406.202,354.814,173.860,47.395,159.581
C06944=1030.988,406.448,354.769,173.872,47.399,159.583
C06945=1030.998,406.693,354.723,173.882,47.403,159.586
C06946=1031.009,406.938,354.678,173.894,47.407,159.588
C06947=1031.019,407.184,354.632,173.904,47.411,159.591
C06948=1031.030,407.430,354.586,173.915,47.415,159.593
C06949=1031.040,407.675,354.541,173.926,47.419,159.596
C06950=1031.050,407.921,354.495,173.937,47.422,159.598
C06951=1031.061,408.166,354.449,173.948,47.427,159.601
C06952=1031.072,408.428,354.400,173.961,47.431,159.604
C06953=1031.083,408.691,354.350,173.972,47.435,159.606
C06954=1031.094,408.953,354.301,173.984,47.440,159.609
C06955=1031.106,409.216,354.252,173.996,47.444,159.612
C06956=1031.116,409.462,354.206,174.007,47.448,159.614
C06957=1031.126,409.707,354.160,174.019,47.452,159.617
C06958=1031.137,409.953,354.114,174.029,47.456,159.619
C06959=1031.148,410.198,354.068,174.041,47.460,159.622
C06960=1031.159,410.443,354.022,174.053,47.464,159.625
C06961=1031.169,410.689,353.976,174.064,47.468,159.627
C06962=1031.179,410.934,353.929,174.075,47.473,159.630
C06963=1031.190,411.180,353.883,174.087,47.477,159.633
C06964=1031.200,411.425,353.835,174.099,47.481,159.635
C06965=1031.211,411.670,353.789,174.110,47.485,159.638
C06966=1031.222,411.916,353.743,174.122,47.490,159.641
C06967=1031.232,412.161,353.696,174.133,47.494,159.643
C06968=1031.243,412.407,353.649,174.144,47.498,159.646
C06969=1031.253,412.653,353.602,174.156,47.502,159.649
C06970=1031.264,412.898,353.556,174.168,47.507,159.652
C06971=1031.274,413.143,353.508,174.180,47.511,159.654
C06972=1031.285,413.388,353.462,174.191,47.515,159.657
C06973=1031.296,413.634,353.414,174.203,47.520,159.660
C06974=1031.307,413.879,353.368,174.215,47.524,159.663
C06975=1031.318,414.124,353.321,174.227,47.529,159.666
C06976=1031.329,414.370,353.273,174.239,47.533,159.668
C06977=1031.340,414.615,353.227,174.251,47.537,159.671
C06978=1031.351,414.861,353.179,174.263,47.542,159.674
C06979=1031.361,415.106,353.132,174.275,47.546,159.677
C06980=1031.372,415.350,353.085,174.287,47.550,159.680
C06981=1031.384,415.596,353.038,174.299,47.555,159.683
C06982=1031.394,415.841,352.990,174.312,47.560,159.686
C06983=1031.406,416.086,352.943,174.324,47.564,159.688
C06984=1031.417,416.332,352.896,174.335,47.569,159.691
C06985=1031.427,416.577,352.848,174.347,47.573,159.694
C06986=1031.438,416.823,352.800,174.361,47.578,159.697
C06987=1031.449,417.068,352.754,174.373,47.583,159.700
C06988=1031.460,417.313,352.705,174.385,47.588,159.703
C06989=1031.471,417.558,352.657,174.397,47.592,159.706
C06990=1031.483,417.803,352.610,174.410,47.597,159.709
C06991=1031.494,418.049,352.562,174.422,47.601,159.712
C06992=1031.505,418.294,352.514,174.434,47.606,159.715
C06993=1031.515,418.539,352.466,174.447,47.611,159.718
C06994=1031.527,418.784,352.418,174.460,47.616,159.721
C06995=1031.538,419.029,352.370,174.473,47.621,159.724
C06996=1031.549,419.275,352.321,174.485,47.625,159.727
C06997=1031.561,419.520,352.274,174.497,47.630,159.730
C06998=1031.571,419.764,352.226,174.510,47.635,159.733
C06999=1031.583,420.010,352.178,174.523,47.640,159.736
C07000=1031.594,420.255,352.129,174.536,47.644,159.739
C07001=1031.606,420.499,352.081,174.550,47.650,159.743
C07002=1031.617,420.745,352.033,174.562,47.655,159.746
C07003=1031.628,420.990,351.984,174.575,47.659,159.749
C07004=1031.640,421.235,351.936,174.587,47.664,159.752
C07005=1031.651,421.480,351.888,174.601,47.669,159.755
C07006=1031.663,421.725,351.839,174.614,47.674,159.758
C07007=1031.674,421.970,351.790,174.627,47.679,159.761
C07008=1031.686,422.215,351.743,174.640,47.684,159.765
C07009=1031.698,422.461,351.693,174.654,47.689,159.768
C07010=1031.709,422.705,351.644,174.666,47.694,159.771
C07011=1031.720,422.951,351.596,174.680,47.699,159.774
C07012=1031.733,423.223,351.541,174.695,47.705,159.778
C07013=1031.746,423.496,351.486,174.710,47.710,159.781
C07014=1031.759,423.768,351.432,174.725,47.716,159.785
C07015=1031.772,424.041,351.377,174.740,47.722,159.789
C07016=1031.784,424.286,351.328,174.753,47.727,159.792
C07017=1031.795,424.531,351.279,174.766,47.732,159.795
C07018=1031.807,424.776,351.230,174.780,47.738,159.799
C07019=1031.819,425.021,351.181,174.794,47.743,159.802
C07020=1031.830,425.266,351.132,174.808,47.748,159.805
C07021=1031.841,425.511,351.083,174.821,47.754,159.809
C07022=1031.854,425.756,351.032,174.835,47.759,159.812
C07023=1031.865,426.000,350.983,174.848,47.764,159.815
C07024=1031.878,426.245,350.934,174.862,47.770,159.819
C07025=1031.890,426.490,350.885,174.877,47.774,159.822
C07026=1031.902,426.735,350.836,174.891,47.780,159.826
C07027=1031.913,426.979,350.786,174.905,47.785,159.829
C07028=1031.926,427.224,350.736,174.919,47.791,159.833
C07029=1031.937,427.470,350.686,174.933,47.796,159.836
C07030=1031.949,427.714,350.636,174.947,47.802,159.840
C07031=1031.961,427.959,350.586,174.962,47.807,159.843
C07032=1031.973,428.203,350.536,174.975,47.813,159.847
C07033=1031.985,428.448,350.486,174.989,47.818,159.850
C07034=1031.996,428.693,350.435,175.004,47.824,159.854
C07035=1032.009,428.938,350.385,175.019,47.830,159.858
C07036=1032.020,429.182,350.336,175.033,47.835,159.861
C07037=1032.033,429.427,350.286,175.048,47.841,159.865
C07038=1032.045,429.671,350.235,175.062,47.846,159.868
C07039=1032.057,429.916,350.184,175.077,47.852,159.872
C07040=1032.069,430.161,350.134,175.091,47.858,159.876
C07041=1032.082,430.406,350.084,175.106,47.863,159.879
C07042=1032.094,430.650,350.033,175.120,47.869,159.883
C07043=1032.107,430.895,349.983,175.135,47.874,159.887
C07044=1032.118,431.139,349.932,175.150,47.881,159.890
C07045=1032.131,431.384,349.881,175.165,47.886,159.894
C07046=1032.143,431.628,349.831,175.180,47.892,159.898
C07047=1032.156,431.873,349.781,175.194,47.898,159.902
C07048=1032.168,432.117,349.730,175.210,47.904,159.905
C07049=1032.181,432.361,349.679,175.225,47.909,159.909
C07050=1032.193,432.606,349.628,175.241,47.915,159.913
C07051=1032.205,432.850,349.577,175.255,47.921,159.917
C07052=1032.218,433.096,349.526,175.270,47.927,159.921
C07053=1032.231,433.340,349.475,175.286,47.933,159.924
C07054=1032.244,433.584,349.425,175.301,47.939,159.928
C07055=1032.256,433.827,349.373,175.317,47.945,159.932
C07056=1032.269,434.073,349.321,175.332,47.951,159.936
C07057=1032.282,434.317,349.271,175.348,47.957,159.940
C07058=1032.294,434.562,349.219,175.363,47.963,159.944
C07059=1032.307,434.806,349.167,175.379,47.969,159.948
C07060=1032.320,435.050,349.116,175.394,47.975,159.952
C07061=1032.332,435.295,349.065,175.410,47.981,159.956
C07062=1032.345,435.539,349.013,175.426,47.987,159.960
C07063=1032.358,435.783,348.961,175.441,47.994,159.964
C07064=1032.370,436.027,348.910,175.458,47.999,159.968
C07065=1032.384,436.272,348.858,175.474,48.006,159.972
C07066=1032.397,436.516,348.805,175.490,48.012,159.976
C07067=1032.410,436.760,348.754,175.505,48.018,159.980
C07068=1032.422,437.005,348.702,175.522,48.024,159.984
C07069=1032.436,437.249,348.650,175.538,48.030,159.988
C07070=1032.448,437.493,348.598,175.554,48.037,159.993
C07071=1032.462,437.737,348.545,175.571,48.043,159.997
C07072=1032.475,437.996,348.490,175.588,48.050,160.001
C07073=1032.489,438.256,348.435,175.606,48.057,160.006
C07074=1032.503,438.516,348.379,175.623,48.063,160.010
C07075=1032.517,438.774,348.323,175.640,48.070,160.015
C07076=1032.530,439.019,348.271,175.657,48.077,160.019
C07077=1032.544,439.263,348.218,175.673,48.083,160.023
C07078=1032.557,439.507,348.166,175.690,48.090,160.028
C07079=1032.570,439.751,348.113,175.708,48.096,160.032
C07080=1032.584,439.995,348.061,175.725,48.103,160.036
C07081=1032.597,440.239,348.008,175.741,48.109,160.040
C07082=1032.610,440.483,347.955,175.758,48.116,160.045
C07083=1032.624,440.727,347.902,175.775,48.123,160.049
C07084=1032.637,440.971,347.849,175.792,48.129,160.054
C07085=1032.651,441.214,347.796,175.810,48.135,160.058
C07086=1032.664,441.458,347.743,175.826,48.142,160.062
C07087=1032.677,441.703,347.690,175.844,48.149,160.067
C07088=1032.691,441.947,347.637,175.861,48.156,160.071
C07089=1032.704,442.191,347.584,175.878,48.162,160.076
C07090=1032.718,442.434,347.531,175.897,48.169,160.080
C07091=1032.732,442.678,347.477,175.914,48.176,160.085
C07092=1032.745,442.922,347.424,175.932,48.183,160.090
C07093=1032.759,443.165,347.370,175.949,48.189,160.094
C07094=1032.773,443.409,347.318,175.967,48.196,160.099
C07095=1032.787,443.653,347.263,175.984,48.203,160.103
C07096=1032.802,443.895,347.211,176.002,48.209,160.108
C07097=1032.817,444.139,347.159,176.020,48.216,160.112
C07098=1032.832,444.382,347.107,176.038,48.223,160.117
C07099=1032.849,444.627,347.055,176.056,48.229,160.122
C07100=1032.865,444.869,347.004,176.074,48.236,160.126
C07101=1032.881,445.113,346.953,176.093,48.242,160.131
C07102=1032.899,445.357,346.903,176.111,48.248,160.135
C07103=1032.917,445.602,346.853,176.130,48.254,160.140
C07104=1032.935,445.845,346.804,176.148,48.260,160.144
C07105=1032.954,446.089,346.755,176.167,48.266,160.149
C07106=1032.974,446.333,346.705,176.185,48.272,160.153
C07107=1032.994,446.577,346.658,176.205,48.278,160.158
C07108=1033.015,446.822,346.610,176.223,48.284,160.162
C07109=1033.036,447.066,346.562,176.242,48.289,160.167
C07110=1033.057,447.310,346.516,176.261,48.295,160.171
C07111=1033.079,447.555,346.469,176.280,48.301,160.176
C07112=1033.102,447.800,346.423,176.299,48.306,160.180
C07113=1033.125,448.044,346.377,176.319,48.312,160.184
C07114=1033.149,448.289,346.331,176.338,48.317,160.189
C07115=1033.173,448.534,346.287,176.358,48.322,160.193
C07116=1033.197,448.779,346.242,176.377,48.327,160.198
C07117=1033.222,449.024,346.198,176.397,48.332,160.202
C07118=1033.248,449.268,346.155,176.417,48.337,160.206
C07119=1033.274,449.514,346.112,176.436,48.342,160.211
C07120=1033.300,449.759,346.069,176.456,48.347,160.215
C07121=1033.328,450.004,346.026,176.475,48.352,160.220
C07122=1033.355,450.250,345.985,176.496,48.357,160.224
C07123=1033.383,450.494,345.943,176.517,48.361,160.229
C07124=1033.412,450.740,345.902,176.536,48.366,160.233
C07125=1033.441,450.986,345.861,176.556,48.370,160.237
C07126=1033.471,451.231,345.821,176.577,48.374,160.241
C07127=1033.501,451.476,345.781,176.598,48.379,160.246
C07128=1033.532,451.722,345.742,176.618,48.383,160.250
C07129=1033.563,451.968,345.703,176.638,48.387,160.254
C07130=1033.595,452.214,345.665,176.659,48.391,160.259
C07131=1033.627,452.458,345.627,176.680,48.396,160.263
C07132=1033.667,452.758,345.581,176.706,48.401,160.268
C07133=1033.707,453.056,345.537,176.732,48.405,160.274
C07134=1033.423,453.120,345.207,176.734,48.472,160.295
C07135=1033.386,452.845,345.248,176.711,48.468,160.290
C07136=1033.349,452.570,345.291,176.687,48.463,160.285
C07137=1033.316,452.324,345.328,176.667,48.459,160.281
C07138=1033.284,452.079,345.366,176.646,48.455,160.276
C07139=1033.252,451.833,345.405,176.625,48.451,160.272
C07140=1033.222,451.586,345.444,176.604,48.447,160.268
C07141=1033.191,451.342,345.483,176.584,48.443,160.264
C07142=1033.161,451.097,345.523,176.563,48.438,160.259
C07143=1033.132,450.851,345.564,176.543,48.434,160.255
C07144=1033.103,450.606,345.604,176.522,48.429,160.250
C07145=1033.074,450.360,345.646,176.502,48.425,160.246
C07146=1033.047,450.116,345.688,176.482,48.421,160.242
C07147=1033.019,449.870,345.729,176.462,48.416,160.237
C07148=1032.992,449.625,345.772,176.442,48.411,160.233
C07149=1032.966,449.380,345.815,176.422,48.406,160.229
C07150=1032.940,449.134,345.858,176.402,48.401,160.224
C07151=1032.914,448.889,345.902,176.382,48.396,160.220
C07152=1032.890,448.644,345.946,176.364,48.392,160.216
C07153=1032.865,448.400,345.991,176.343,48.387,160.211
C07154=1032.841,448.155,346.036,176.324,48.381,160.207
C07155=1032.818,447.910,346.081,176.304,48.376,160.202
C07156=1032.795,447.666,346.128,176.285,48.371,160.198
C07157=1032.773,447.421,346.173,176.266,48.365,160.193
C07158=1032.750,447.176,346.220,176.247,48.360,160.189
C07159=1032.730,446.932,346.268,176.228,48.355,160.184
C07160=1032.709,446.688,346.315,176.210,48.349,160.180
C07161=1032.678,446.313,346.389,176.180,48.340,160.173
C07162=1032.648,445.939,346.463,176.151,48.331,160.166
C07163=1032.620,445.566,346.538,176.123,48.322,160.159
C07164=1032.592,445.193,346.615,176.095,48.313,160.152
C07165=1032.574,444.949,346.666,176.077,48.306,160.148
C07166=1032.558,444.706,346.717,176.058,48.300,160.143
C07167=1032.542,444.462,346.769,176.040,48.294,160.139
C07168=1032.527,444.219,346.820,176.021,48.288,160.134
C07169=1032.511,443.975,346.872,176.004,48.281,160.130
C07170=1032.497,443.731,346.924,175.985,48.274,160.125
C07171=1032.483,443.488,346.978,175.968,48.268,160.120
C07172=1032.469,443.245,347.031,175.950,48.261,160.116
C07173=1032.454,443.002,347.084,175.933,48.254,160.111
C07174=1032.441,442.758,347.138,175.915,48.248,160.107
C07175=1032.427,442.515,347.191,175.897,48.241,160.102
C07176=1032.413,442.271,347.245,175.880,48.234,160.098
C07177=1032.400,442.026,347.298,175.862,48.228,160.093
C07178=1032.386,441.782,347.351,175.845,48.221,160.089
C07179=1032.373,441.538,347.404,175.827,48.214,160.084
C07180=1032.359,441.295,347.457,175.810,48.208,160.080
C07181=1032.345,441.050,347.510,175.793,48.201,160.075
C07182=1032.332,440.806,347.563,175.776,48.195,160.071
C07183=1032.318,440.562,347.616,175.759,48.189,160.067
C07184=1032.305,440.318,347.669,175.741,48.182,160.062
C07185=1032.291,440.075,347.722,175.725,48.175,160.058
C07186=1032.278,439.831,347.775,175.708,48.169,160.053
C07187=1032.266,439.586,347.827,175.691,48.162,160.049
C07188=1032.252,439.343,347.880,175.674,48.157,160.045
C07189=1032.231,438.968,347.960,175.648,48.146,160.038
C07190=1032.211,438.593,348.041,175.623,48.137,160.032
C07191=1032.191,438.219,348.121,175.597,48.127,160.025
C07192=1032.171,437.843,348.201,175.572,48.117,160.019
C07193=1032.158,437.599,348.253,175.556,48.111,160.015
C07194=1032.145,437.355,348.306,175.539,48.105,160.011
C07195=1032.132,437.111,348.357,175.523,48.099,160.007
C07196=1032.119,436.866,348.410,175.507,48.092,160.002
C07197=1032.106,436.622,348.462,175.491,48.086,159.998
C07198=1032.094,436.378,348.514,175.475,48.080,159.994
C07199=1032.080,436.134,348.566,175.459,48.074,159.990
C07200=1032.067,435.890,348.616,175.443,48.069,159.986
C07201=1032.055,435.645,348.669,175.427,48.062,159.982
C07202=1032.042,435.402,348.720,175.411,48.056,159.978
C07203=1032.028,435.157,348.772,175.395,48.050,159.974
C07204=1032.016,434.913,348.824,175.380,48.044,159.970
C07205=1032.003,434.668,348.875,175.364,48.038,159.966
C07206=1031.991,434.423,348.926,175.349,48.032,159.962
C07207=1031.978,434.179,348.978,175.332,48.026,159.958
C07208=1031.965,433.935,349.029,175.317,48.020,159.954
C07209=1031.953,433.690,349.080,175.301,48.015,159.950
C07210=1031.940,433.445,349.132,175.286,48.009,159.947
C07211=1031.927,433.201,349.182,175.271,48.002,159.943
C07212=1031.914,432.956,349.234,175.256,47.996,159.939
C07213=1031.901,432.712,349.284,175.240,47.991,159.935
C07214=1031.890,432.468,349.336,175.225,47.985,159.931
C07215=1031.877,432.223,349.386,175.210,47.980,159.927
C07216=1031.865,431.979,349.437,175.194,47.974,159.924
C07217=1031.852,431.734,349.488,175.180,47.968,159.920
C07218=1031.840,431.490,349.538,175.165,47.963,159.916
C07219=1031.827,431.245,349.589,175.150,47.957,159.912
C07220=1031.815,431.000,349.640,175.134,47.951,159.909
C07221=1031.802,430.755,349.690,175.120,47.945,159.905
C07222=1031.791,430.511,349.740,175.105,47.940,159.901
C07223=1031.778,430.267,349.791,175.091,47.934,159.898
C07224=1031.766,430.022,349.841,175.076,47.929,159.894
C07225=1031.754,429.777,349.892,175.062,47.923,159.890
C07226=1031.741,429.533,349.942,175.046,47.917,159.887
C07227=1031.729,429.288,349.993,175.032,47.912,159.883
C07228=1031.717,429.043,350.043,175.017,47.906,159.879
C07229=1031.705,428.799,350.092,175.003,47.901,159.876
C07230=1031.693,428.554,350.143,174.988,47.895,159.872
C07231=1031.681,428.309,350.193,174.974,47.890,159.869
C07232=1031.669,428.064,350.243,174.960,47.884,159.865
C07233=1031.657,427.820,350.293,174.946,47.879,159.862
C07234=1031.645,427.575,350.343,174.932,47.874,159.858
C07235=1031.634,427.331,350.392,174.917,47.868,159.855
C07236=1031.622,427.086,350.443,174.904,47.863,159.851
C07237=1031.610,426.841,350.493,174.889,47.858,159.848
C07238=1031.598,426.596,350.542,174.875,47.853,159.844
C07239=1031.586,426.351,350.592,174.861,47.847,159.841
C07240=1031.574,426.106,350.641,174.847,47.842,159.837
C07241=1031.562,425.861,350.690,174.834,47.837,159.834
C07242=1031.549,425.616,350.740,174.820,47.831,159.831
C07243=1031.538,425.372,350.789,174.805,47.826,159.827
C07244=1031.527,425.127,350.838,174.791,47.821,159.824
C07245=1031.515,424.882,350.887,174.778,47.816,159.820
C07246=1031.503,424.637,350.937,174.764,47.811,159.817
C07247=1031.492,424.393,350.986,174.750,47.806,159.814
C07248=1031.480,424.147,351.035,174.737,47.800,159.810
C07249=1031.467,423.873,351.090,174.722,47.795,159.807
C07250=1031.454,423.598,351.146,174.707,47.789,159.803
C07251=1031.441,423.323,351.201,174.692,47.784,159.800
C07252=1031.428,423.048,351.255,174.677,47.777,159.796
C07253=1031.417,422.803,351.304,174.664,47.773,159.793
C07254=1031.405,422.558,351.353,174.650,47.768,159.789
C07255=1031.393,422.312,351.401,174.637,47.763,159.786
C07256=1031.382,422.068,351.450,174.623,47.758,159.783
C07257=1031.370,421.823,351.498,174.611,47.753,159.780
C07258=1031.358,421.578,351.547,174.598,47.748,159.777
C07259=1031.347,421.332,351.595,174.584,47.743,159.773
C07260=1031.336,421.088,351.644,174.572,47.738,159.770
C07261=1031.324,420.843,351.692,174.558,47.733,159.767
C07262=1031.313,420.597,351.740,174.545,47.729,159.764
C07263=1031.301,420.353,351.789,174.533,47.724,159.761
C07264=1031.290,420.108,351.837,174.520,47.719,159.758
C07265=1031.279,419.862,351.885,174.506,47.714,159.755
C07266=1031.267,419.617,351.934,174.494,47.709,159.752
C07267=1031.256,419.371,351.982,174.481,47.705,159.749
C07268=1031.245,419.127,352.029,174.468,47.700,159.746
C07269=1031.234,418.882,352.078,174.455,47.696,159.743
C07270=1031.223,418.636,352.126,174.443,47.691,159.740
C07271=1031.211,418.391,352.174,174.431,47.686,159.736
C07272=1031.201,418.147,352.222,174.418,47.682,159.734
C07273=1031.189,417.901,352.270,174.406,47.677,159.731
C07274=1031.178,417.656,352.317,174.393,47.672,159.728
C07275=1031.167,417.411,352.365,174.380,47.667,159.725
